(* CODESYS project PRG1545637205.project

Project tree, tasks and I/O mapping:
  Device : CODESYS Control for Raspberry Pi, 3S - Smart Software Solutions GmbH, version 3.5.7.10
    application Application
      libraries: Standard, * (System); SysSocket, 3.5.9.0 (System); SysSem, 3.5.5.0 (System); SysCom, 3.5.5.0 (System); Util, 3.5.11.0 (System); MQTT Client Library, 3.5.0.0 (Stefan Roßmann Engineering Solutions); SysTimeRtc, * (System)
      task MainTask (cyclic, interval t#20ms, priority 1) calls PLC_PRG, Cement_PRG, Automode, Formula, LimeSand, Mixer_PRG, Logger
      task VISU_TASK (cyclic, interval 100 ms, priority 31) calls VisuElems.Visu_Prg
      program PLC_PRG [ST]
      vis/
        visualisation Visualization
        visualisation formula
        visualisation packing
        visualisation lime
        visualisation cement
        visualisation mixer
        visualisation dust
        visualisation other
        visualisation cement_1
        visualisation cement_0
        visualisation cement_2
        visualisation lime_0
        visualisation lime_1
        visualisation lime_3
        visualisation lime_2
        visualisation cement_3
        visualisation mixer_0
        visualisation mixer_1
        visualisation mixer_2
        visualisation mixer_3
        visualisation packing_0
        visualisation packing_3
        visualisation packing_2
        visualisation packing_1
      function block INVT_AO [LD]
      function block Constancheck [ST]
      function block ParamAdjust [ST]
      program LimeSand [LD]
      function block interupt [LD]
      function block Alarm [ST]
      program Automode [LD]
      function block BAYKON [LD]
      program Cement_PRG [LD]
      program Formula [LD]
      function block Formula_Loader [ST]
      function block PulseHold [LD]
      function block screw_speed [ST]
      program Mixer_PRG [LD]
      function block Cycletime [LD]
      MYSQL/
        DUTs/
          data type SHA1Context
          data type MySql_FieldInfo
          data type MySql_FieldTypes
          data type MySql_ResultSet
          data type MySql_ServerInfo
        private/
          SHA/
            function SHA1Hex2String [ST]
            function SHA1Input [ST]
            function SHA1PadMessage [ST]
            function SHA1ProcessMessageBlock [ST]
            function SHA1Reset [ST]
            function SHA1Result [ST]
            function SHA1Version [ST]
            function SHA1 [ST]
          function MySql_Close [ST]
          function block MySql_Context [ST]
          function MySql_Scramble [ST]
        public/
          function MySql_GetStringValue [ST]
          function MySql_Version [ST]
          function block MySql_Execute [ST]
          function block MySql_Login [ST]
          function block MySql_Logout [ST]
          function block MySql_Query [ST]
      global variables GVL_MYSQL
      function block DC [LD]
      program Logger [ST]
    SoftMotion General Axis Pool
    I²C
    SPI
    GPIOs_A_B : GPIOs A/B, 3S - Smart Software Solutions GmbH, version 1.1.1.10
        unmapped channels: digital inputs (GPIO0..GPIO31), digital outputs (GPIO0..GPIO31)
    Onewire
    Camera device
      <Empty>
    Ethernet : Ethernet, 3S - Smart Software Solutions GmbH, version 3.5.10.0
      Modbus_TCP_Master : Modbus TCP Master, 3S - Smart Software Solutions GmbH, version 3.5.10.0
          settings: AutoReconnect = TRUE
        WAGO_170 : Modbus TCP Slave, 3S - Smart Software Solutions GmbH, version 3.5.10.0
            settings: IPAddress = [192, 168, 100, 170]; Channel 0.Function Code = 2; Channel 0.Read Offset = 16#0000; Channel 0.Read Length = 128; Channel 0.Write Offset = 0; Channel 0.Write Length = 0; Channel 0.Cycle Time = 100; Channel 1.Function Code = 3; Channel 1.Read Offset = 16#0000; Channel 1.Read Length = 8; Channel 1.Write Offset = 0; Channel 1.Write Length = 0; Channel 1.Cycle Time = 100; Channel 2.Function Code = 15; Channel 2.Read Offset = 0; Channel 2.Read Length = 0; Channel 2.Write Offset = 16#0000; Channel 2.Write Length = 80; Channel 2.Cycle Time = 100; Channel 3.Function Code = 16; Channel 3.Read Offset = 0; Channel 3.Read Length = 0; Channel 3.Write Offset = 16#0000; Channel 3.Write Length = 4; Channel 3.Cycle Time = 100
            input  DI : ARRAY[0..15] OF BYTE  // Channel 0
            input  DI120 : BYTE  // Channel 0.Channel 0
            input  DI121 : BOOL  // Channel 0.Channel 0.Bit0
            input  DI122 : BOOL  // Channel 0.Channel 0.Bit1
            input  DI123 : BOOL  // Channel 0.Channel 0.Bit2
            input  DI124 : BOOL  // Channel 0.Channel 0.Bit3
            input  DI125 : BOOL  // Channel 0.Channel 0.Bit4
            input  DI126 : BOOL  // Channel 0.Channel 0.Bit5
            input  DI127 : BOOL  // Channel 0.Channel 0.Bit6
            input  DI128 : BOOL  // Channel 0.Channel 0.Bit7
            input  DI130 : BYTE  // Channel 0.Channel 0
            input  DI131 : BOOL  // Channel 0.Channel 0.Bit0
            input  DI132 : BOOL  // Channel 0.Channel 0.Bit1
            input  DI133 : BOOL  // Channel 0.Channel 0.Bit2
            input  DI134 : BOOL  // Channel 0.Channel 0.Bit3
            input  DI135 : BOOL  // Channel 0.Channel 0.Bit4
            input  DI136 : BOOL  // Channel 0.Channel 0.Bit5
            input  DI137 : BOOL  // Channel 0.Channel 0.Bit6
            input  DI138 : BOOL  // Channel 0.Channel 0.Bit7
            input  DI140 : BYTE  // Channel 0.Channel 0
            input  DI141 : BOOL  // Channel 0.Channel 0.Bit0
            input  DI142 : BOOL  // Channel 0.Channel 0.Bit1
            input  DI143 : BOOL  // Channel 0.Channel 0.Bit2
            input  DI144 : BOOL  // Channel 0.Channel 0.Bit3
            input  DI145 : BOOL  // Channel 0.Channel 0.Bit4
            input  DI146 : BOOL  // Channel 0.Channel 0.Bit5
            input  DI147 : BOOL  // Channel 0.Channel 0.Bit6
            input  DI148 : BOOL  // Channel 0.Channel 0.Bit7
            input  DI150 : BYTE  // Channel 0.Channel 0
            input  DI151 : BOOL  // Channel 0.Channel 0.Bit0
            input  DI152 : BOOL  // Channel 0.Channel 0.Bit1
            input  DI153 : BOOL  // Channel 0.Channel 0.Bit2
            input  DI154 : BOOL  // Channel 0.Channel 0.Bit3
            input  DI155 : BOOL  // Channel 0.Channel 0.Bit4
            input  DI156 : BOOL  // Channel 0.Channel 0.Bit5
            input  DI157 : BOOL  // Channel 0.Channel 0.Bit6
            input  DI158 : BOOL  // Channel 0.Channel 0.Bit7
            input  DI160 : BYTE  // Channel 0.Channel 0
            input  DI161 : BOOL  // Channel 0.Channel 0.Bit0
            input  DI162 : BOOL  // Channel 0.Channel 0.Bit1
            input  DI163 : BOOL  // Channel 0.Channel 0.Bit2
            input  DI164 : BOOL  // Channel 0.Channel 0.Bit3
            input  DI165 : BOOL  // Channel 0.Channel 0.Bit4
            input  DI166 : BOOL  // Channel 0.Channel 0.Bit5
            input  DI167 : BOOL  // Channel 0.Channel 0.Bit6
            input  DI168 : BOOL  // Channel 0.Channel 0.Bit7
            input  DI170 : BYTE  // Channel 0.Channel 0
            input  DI171 : BOOL  // Channel 0.Channel 0.Bit0
            input  DI172 : BOOL  // Channel 0.Channel 0.Bit1
            input  DI173 : BOOL  // Channel 0.Channel 0.Bit2
            input  DI174 : BOOL  // Channel 0.Channel 0.Bit3
            input  DI175 : BOOL  // Channel 0.Channel 0.Bit4
            input  DI176 : BOOL  // Channel 0.Channel 0.Bit5
            input  DI177 : BOOL  // Channel 0.Channel 0.Bit6
            input  DI178 : BOOL  // Channel 0.Channel 0.Bit7
            input  DI180 : BYTE  // Channel 0.Channel 0
            input  DI181 : BOOL  // Channel 0.Channel 0.Bit0
            input  DI182 : BOOL  // Channel 0.Channel 0.Bit1
            input  DI183 : BOOL  // Channel 0.Channel 0.Bit2
            input  DI184 : BOOL  // Channel 0.Channel 0.Bit3
            input  DI185 : BOOL  // Channel 0.Channel 0.Bit4
            input  DI186 : BOOL  // Channel 0.Channel 0.Bit5
            input  DI187 : BOOL  // Channel 0.Channel 0.Bit6
            input  DI188 : BOOL  // Channel 0.Channel 0.Bit7
            input  DI190 : BYTE  // Channel 0.Channel 0
            input  DI191 : BOOL  // Channel 0.Channel 0.Bit0
            input  DI192 : BOOL  // Channel 0.Channel 0.Bit1
            input  DI193 : BOOL  // Channel 0.Channel 0.Bit2
            input  DI194 : BOOL  // Channel 0.Channel 0.Bit3
            input  DI195 : BOOL  // Channel 0.Channel 0.Bit4
            input  DI196 : BOOL  // Channel 0.Channel 0.Bit5
            input  DI197 : BOOL  // Channel 0.Channel 0.Bit6
            input  DI198 : BOOL  // Channel 0.Channel 0.Bit7
            input  DI200 : BYTE  // Channel 0.Channel 0
            input  DI201 : BOOL  // Channel 0.Channel 0.Bit0
            input  DI202 : BOOL  // Channel 0.Channel 0.Bit1
            input  DI203 : BOOL  // Channel 0.Channel 0.Bit2
            input  DI204 : BOOL  // Channel 0.Channel 0.Bit3
            input  DI205 : BOOL  // Channel 0.Channel 0.Bit4
            input  DI206 : BOOL  // Channel 0.Channel 0.Bit5
            input  DI207 : BOOL  // Channel 0.Channel 0.Bit6
            input  DI208 : BOOL  // Channel 0.Channel 0.Bit7
            input  DI210 : BYTE  // Channel 0.Channel 0
            input  DI211 : BOOL  // Channel 0.Channel 0.Bit0
            input  DI212 : BOOL  // Channel 0.Channel 0.Bit1
            input  DI213 : BOOL  // Channel 0.Channel 0.Bit2
            input  DI214 : BOOL  // Channel 0.Channel 0.Bit3
            input  DI215 : BOOL  // Channel 0.Channel 0.Bit4
            input  DI216 : BOOL  // Channel 0.Channel 0.Bit5
            input  DI217 : BOOL  // Channel 0.Channel 0.Bit6
            input  DI218 : BOOL  // Channel 0.Channel 0.Bit7
            input  DI220 : BYTE  // Channel 0.Channel 0
            input  DI221 : BOOL  // Channel 0.Channel 0.Bit0
            input  DI222 : BOOL  // Channel 0.Channel 0.Bit1
            input  DI223 : BOOL  // Channel 0.Channel 0.Bit2
            input  DI224 : BOOL  // Channel 0.Channel 0.Bit3
            input  DI225 : BOOL  // Channel 0.Channel 0.Bit4
            input  DI226 : BOOL  // Channel 0.Channel 0.Bit5
            input  DI227 : BOOL  // Channel 0.Channel 0.Bit6
            input  DI228 : BOOL  // Channel 0.Channel 0.Bit7
            input  DI230 : BYTE  // Channel 0.Channel 0
            input  DI231 : BOOL  // Channel 0.Channel 0.Bit0
            input  DI232 : BOOL  // Channel 0.Channel 0.Bit1
            input  DI233 : BOOL  // Channel 0.Channel 0.Bit2
            input  DI234 : BOOL  // Channel 0.Channel 0.Bit3
            input  DI235 : BOOL  // Channel 0.Channel 0.Bit4
            input  DI236 : BOOL  // Channel 0.Channel 0.Bit5
            input  DI237 : BOOL  // Channel 0.Channel 0.Bit6
            input  DI238 : BOOL  // Channel 0.Channel 0.Bit7
            input  DI240 : BYTE  // Channel 0.Channel 0
            input  DI241 : BOOL  // Channel 0.Channel 0.Bit0
            input  DI242 : BOOL  // Channel 0.Channel 0.Bit1
            input  DI243 : BOOL  // Channel 0.Channel 0.Bit2
            input  DI244 : BOOL  // Channel 0.Channel 0.Bit3
            input  DI245 : BOOL  // Channel 0.Channel 0.Bit4
            input  DI246 : BOOL  // Channel 0.Channel 0.Bit5
            input  DI247 : BOOL  // Channel 0.Channel 0.Bit6
            input  DI248 : BOOL  // Channel 0.Channel 0.Bit7
            input  DI250 : BYTE  // Channel 0.Channel 0
            input  DI251 : BOOL  // Channel 0.Channel 0.Bit0
            input  DI252 : BOOL  // Channel 0.Channel 0.Bit1
            input  DI253 : BOOL  // Channel 0.Channel 0.Bit2
            input  DI254 : BOOL  // Channel 0.Channel 0.Bit3
            input  DI255 : BOOL  // Channel 0.Channel 0.Bit4
            input  DI256 : BOOL  // Channel 0.Channel 0.Bit5
            input  DI257 : BOOL  // Channel 0.Channel 0.Bit6
            input  DI258 : BOOL  // Channel 0.Channel 0.Bit7
            input  DI260 : BYTE  // Channel 0.Channel 0
            input  DI261 : BOOL  // Channel 0.Channel 0.Bit0
            input  DI262 : BOOL  // Channel 0.Channel 0.Bit1
            input  DI263 : BOOL  // Channel 0.Channel 0.Bit2
            input  DI264 : BOOL  // Channel 0.Channel 0.Bit3
            input  DI265 : BOOL  // Channel 0.Channel 0.Bit4
            input  DI266 : BOOL  // Channel 0.Channel 0.Bit5
            input  DI267 : BOOL  // Channel 0.Channel 0.Bit6
            input  DI268 : BOOL  // Channel 0.Channel 0.Bit7
            input  DI270 : BYTE  // Channel 0.Channel 0
            input  DI271 : BOOL  // Channel 0.Channel 0.Bit0
            input  DI272 : BOOL  // Channel 0.Channel 0.Bit1
            input  DI273 : BOOL  // Channel 0.Channel 0.Bit2
            input  DI274 : BOOL  // Channel 0.Channel 0.Bit3
            input  DI275 : BOOL  // Channel 0.Channel 0.Bit4
            input  DI276 : BOOL  // Channel 0.Channel 0.Bit5
            input  DI277 : BOOL  // Channel 0.Channel 0.Bit6
            input  DI278 : BOOL  // Channel 0.Channel 0.Bit7
            input  AI : ARRAY[0..7] OF WORD  // Channel 1
            input  AI281 : WORD  // Channel 1.Channel 1
            input  AI282 : WORD  // Channel 1.Channel 1
            input  AI283 : WORD  // Channel 1.Channel 1
            input  AI284 : WORD  // Channel 1.Channel 1
            input  AI291 : WORD  // Channel 1.Channel 1
            input  AI292 : WORD  // Channel 1.Channel 1
            input  AI293 : WORD  // Channel 1.Channel 1
            input  AI294 : WORD  // Channel 1.Channel 1
            output DO311 : BOOL  // Channel 2.Channel 2.Bit0
            output DO312 : BOOL  // Channel 2.Channel 2.Bit1
            output DO313 : BOOL  // Channel 2.Channel 2.Bit2
            output DO314 : BOOL  // Channel 2.Channel 2.Bit3
            output DO315 : BOOL  // Channel 2.Channel 2.Bit4
            output DO316 : BOOL  // Channel 2.Channel 2.Bit5
            output DO317 : BOOL  // Channel 2.Channel 2.Bit6
            output DO318 : BOOL  // Channel 2.Channel 2.Bit7
            output DO321 : BOOL  // Channel 2.Channel 2.Bit0
            output DO322 : BOOL  // Channel 2.Channel 2.Bit1
            output DO323 : BOOL  // Channel 2.Channel 2.Bit2
            output DO324 : BOOL  // Channel 2.Channel 2.Bit3
            output DO325 : BOOL  // Channel 2.Channel 2.Bit4
            output DO326 : BOOL  // Channel 2.Channel 2.Bit5
            output DO327 : BOOL  // Channel 2.Channel 2.Bit6
            output DO328 : BOOL  // Channel 2.Channel 2.Bit7
            output DO331 : BOOL  // Channel 2.Channel 2.Bit0
            output DO332 : BOOL  // Channel 2.Channel 2.Bit1
            output DO333 : BOOL  // Channel 2.Channel 2.Bit2
            output DO334 : BOOL  // Channel 2.Channel 2.Bit3
            output DO335 : BOOL  // Channel 2.Channel 2.Bit4
            output DO336 : BOOL  // Channel 2.Channel 2.Bit5
            output DO337 : BOOL  // Channel 2.Channel 2.Bit6
            output DO338 : BOOL  // Channel 2.Channel 2.Bit7
            output DO341 : BOOL  // Channel 2.Channel 2.Bit0
            output DO342 : BOOL  // Channel 2.Channel 2.Bit1
            output DO343 : BOOL  // Channel 2.Channel 2.Bit2
            output DO344 : BOOL  // Channel 2.Channel 2.Bit3
            output DO345 : BOOL  // Channel 2.Channel 2.Bit4
            output DO346 : BOOL  // Channel 2.Channel 2.Bit5
            output DO347 : BOOL  // Channel 2.Channel 2.Bit6
            output DO348 : BOOL  // Channel 2.Channel 2.Bit7
            output DO351 : BOOL  // Channel 2.Channel 2.Bit0
            output DO352 : BOOL  // Channel 2.Channel 2.Bit1
            output DO353 : BOOL  // Channel 2.Channel 2.Bit2
            output DO354 : BOOL  // Channel 2.Channel 2.Bit3
            output DO355 : BOOL  // Channel 2.Channel 2.Bit4
            output DO356 : BOOL  // Channel 2.Channel 2.Bit5
            output DO357 : BOOL  // Channel 2.Channel 2.Bit6
            output DO358 : BOOL  // Channel 2.Channel 2.Bit7
            output DO371 : BOOL  // Channel 2.Channel 2.Bit0
            output DO372 : BOOL  // Channel 2.Channel 2.Bit1
            output DO373 : BOOL  // Channel 2.Channel 2.Bit2
            output DO374 : BOOL  // Channel 2.Channel 2.Bit3
            output DO375 : BOOL  // Channel 2.Channel 2.Bit4
            output DO376 : BOOL  // Channel 2.Channel 2.Bit5
            output DO377 : BOOL  // Channel 2.Channel 2.Bit6
            output DO378 : BOOL  // Channel 2.Channel 2.Bit7
            output DO381 : BOOL  // Channel 2.Channel 2.Bit0
            output DO382 : BOOL  // Channel 2.Channel 2.Bit1
            output DO383 : BOOL  // Channel 2.Channel 2.Bit2
            output DO384 : BOOL  // Channel 2.Channel 2.Bit3
            output DO385 : BOOL  // Channel 2.Channel 2.Bit4
            output DO386 : BOOL  // Channel 2.Channel 2.Bit5
            output DO387 : BOOL  // Channel 2.Channel 2.Bit6
            output DO388 : BOOL  // Channel 2.Channel 2.Bit7
            output DO391 : BOOL  // Channel 2.Channel 2.Bit0
            output DO392 : BOOL  // Channel 2.Channel 2.Bit1
            output DO393 : BOOL  // Channel 2.Channel 2.Bit2
            output DO394 : BOOL  // Channel 2.Channel 2.Bit3
            output DO395 : BOOL  // Channel 2.Channel 2.Bit4
            output DO396 : BOOL  // Channel 2.Channel 2.Bit5
            output DO397 : BOOL  // Channel 2.Channel 2.Bit6
            output DO398 : BOOL  // Channel 2.Channel 2.Bit7
            output DO401 : BOOL  // Channel 2.Channel 2.Bit0
            output DO402 : BOOL  // Channel 2.Channel 2.Bit1
            output DO403 : BOOL  // Channel 2.Channel 2.Bit2
            output DO404 : BOOL  // Channel 2.Channel 2.Bit3
            output DO405 : BOOL  // Channel 2.Channel 2.Bit4
            output DO406 : BOOL  // Channel 2.Channel 2.Bit5
            output DO407 : BOOL  // Channel 2.Channel 2.Bit6
            output DO408 : BOOL  // Channel 2.Channel 2.Bit7
            output DO411 : BOOL  // Channel 2.Channel 2.Bit0
            output DO412 : BOOL  // Channel 2.Channel 2.Bit1
            output DO413 : BOOL  // Channel 2.Channel 2.Bit2
            output DO414 : BOOL  // Channel 2.Channel 2.Bit3
            output DO415 : BOOL  // Channel 2.Channel 2.Bit4
            output DO416 : BOOL  // Channel 2.Channel 2.Bit5
            output DO417 : BOOL  // Channel 2.Channel 2.Bit6
            output DO418 : BOOL  // Channel 2.Channel 2.Bit7
            output AO431 : WORD  // Channel 3.Channel 3
            output AO432 : WORD  // Channel 3.Channel 3
            output AO441 : WORD  // Channel 3.Channel 3
            output AO442 : WORD  // Channel 3.Channel 3
            unmapped channels: Channel 2, Channel 3
        Baykon_171 : Modbus TCP Slave, 3S - Smart Software Solutions GmbH, version 3.5.10.0
            settings: Unit-ID = 1; IPAddress = [192, 168, 100, 171]; Channel 0.Function Code = 3; Channel 0.Read Offset = 16#0000; Channel 0.Read Length = 7; Channel 0.Write Offset = 0; Channel 0.Write Length = 0; Channel 0.Cycle Time = 100
            input  cem1 : WORD  // Channel 0.Channel 0
            input  cem2 : WORD  // Channel 0.Channel 0
            input  cem3 : WORD  // Channel 0.Channel 0
            input  cem4 : WORD  // Channel 0.Channel 0
            input  cem5 : WORD  // Channel 0.Channel 0
            input  cem6 : WORD  // Channel 0.Channel 0
            input  cem7 : WORD  // Channel 0.Channel 0
            unmapped channels: Channel 0
        Baykon_172 : Modbus TCP Slave, 3S - Smart Software Solutions GmbH, version 3.5.10.0
            settings: Unit-ID = 1; IPAddress = [192, 168, 100, 172]; Channel 0.Function Code = 3; Channel 0.Read Offset = 16#0000; Channel 0.Read Length = 7; Channel 0.Write Offset = 0; Channel 0.Write Length = 0; Channel 0.Cycle Time = 100
            input  lime1 : WORD  // Channel 0.Channel 0
            input  lime2 : WORD  // Channel 0.Channel 0
            input  lime3 : WORD  // Channel 0.Channel 0
            input  lime4 : WORD  // Channel 0.Channel 0
            input  lime5 : WORD  // Channel 0.Channel 0
            input  lime6 : WORD  // Channel 0.Channel 0
            input  lime7 : WORD  // Channel 0.Channel 0
            unmapped channels: Channel 0
  libraries: VisuSymbols, 3.5.10.0 (System)
  text list GlobalTextList
*)

// Device/Application/MYSQL/DUTs/SHA1Context
TYPE SHA1Context :
(* This structure will hold context information for the hashing operation *)
  STRUCT
	Message_Digest : ARRAY [0..4] OF DWORD ;(* Message Digest (output)          *)
    Length_Low  : DWORD;        			(* Message length in bits           *)
    Length_High : DWORD;       				(* Message length in bits           *)
    Message_Block : ARRAY [0..63] OF BYTE; 	(* 512-bit message blocks      *)
    Message_Block_Index : INT;    			(* Index into message block array   *)
    Computed : BOOL;               			(* Is the digest computed?          *)
    Corrupted: BOOL;              			(* Is the message digest corruped?  *)
  END_STRUCT
END_TYPE

// Device/Application/MYSQL/DUTs/MySql_FieldInfo
TYPE MySql_FieldInfo :
(* This structure contains detail informations about each "column" or "data field" in a result set *)
  STRUCT
	sName : STRING(gcMySql_dwMaxIdentifierLength);
	udiLength : UDINT;
	eType : MySql_FieldTypes;
	wFlags : WORD;
	bDecimals : BYTE;
  END_STRUCT
END_TYPE

(*
VERSION 4.1
 Bytes                      Name
 -----                      ----
 n (Length Coded String)    catalog
 n (Length Coded String)    db
 n (Length Coded String)    table
 n (Length Coded String)    org_table
 n (Length Coded String)    name
 n (Length Coded String)    org_name
 1                          (filler)
 2                          charsetnr
 4                          length
 1                          type
 2                          flags
 1                          decimals
 2                          (filler), always 0x00
 n (Length Coded Binary)    default


length:                  Length of column, according to the definition.
                         Also known as "display length". The value given
                         here may be larger than the actual length, for
                         example an instance of a VARCHAR(2) column may
                         have only 1 character in it.

type:                    The code for the column's data type. Also known as
                         "enum_field_type". The possible values at time of
                         writing (taken from  include/mysql_com.h), in hexadecimal:
                         0x00   FIELD_TYPE_DECIMAL
                         0x01   FIELD_TYPE_TINY
                         0x02   FIELD_TYPE_SHORT
                         0x03   FIELD_TYPE_LONG
                         0x04   FIELD_TYPE_FLOAT
                         0x05   FIELD_TYPE_DOUBLE
                         0x06   FIELD_TYPE_NULL
                         0x07   FIELD_TYPE_TIMESTAMP
                         0x08   FIELD_TYPE_LONGLONG
                         0x09   FIELD_TYPE_INT24
                         0x0a   FIELD_TYPE_DATE
                         0x0b   FIELD_TYPE_TIME
                         0x0c   FIELD_TYPE_DATETIME
                         0x0d   FIELD_TYPE_YEAR
                         0x0e   FIELD_TYPE_NEWDATE
                         0x0f   FIELD_TYPE_VARCHAR (new in MySQL 5.0)
                         0x10   FIELD_TYPE_BIT (new in MySQL 5.0)
                         0xf6   FIELD_TYPE_NEWDECIMAL (new in MYSQL 5.0)
                         0xf7   FIELD_TYPE_ENUM
                         0xf8   FIELD_TYPE_SET
                         0xf9   FIELD_TYPE_TINY_BLOB
                         0xfa   FIELD_TYPE_MEDIUM_BLOB
                         0xfb   FIELD_TYPE_LONG_BLOB
                         0xfc   FIELD_TYPE_BLOB
                         0xfd   FIELD_TYPE_VAR_STRING
                         0xfe   FIELD_TYPE_STRING
                         0xff   FIELD_TYPE_GEOMETRY

flags:                   The possible flag values at time of
                         writing (taken from  include/mysql_com.h), in hexadecimal:
                         0001 NOT_NULL_FLAG
                         0002 PRI_KEY_FLAG
                         0004 UNIQUE_KEY_FLAG
                         0008 MULTIPLE_KEY_FLAG
                         0010 BLOB_FLAG
                         0020 UNSIGNED_FLAG
                         0040 ZEROFILL_FLAG
                         0080 BINARY_FLAG
                         0100 ENUM_FLAG
                         0200 AUTO_INCREMENT_FLAG
                         0400 TIMESTAMP_FLAG
                         0800 SET_FLAG

decimals:                The number of positions after the decimal
                         point if the type is DECIMAL or NUMERIC.
                         Also known as "scale".


*)

// Device/Application/MYSQL/DUTs/MySql_FieldTypes
TYPE MySql_FieldTypes :
(
	MYSQL_TYPE_DECIMAL,
	MYSQL_TYPE_TINY,
	MYSQL_TYPE_SHORT,
	MYSQL_TYPE_LONG,
	MYSQL_TYPE_FLOAT,
	MYSQL_TYPE_DOUBLE,
	MYSQL_TYPE_NULL,
	MYSQL_TYPE_TIMESTAMP,
	MYSQL_TYPE_LONGLONG,
	MYSQL_TYPE_INT24,
	MYSQL_TYPE_DATE,
	MYSQL_TYPE_TIME,
	MYSQL_TYPE_DATETIME,
	MYSQL_TYPE_YEAR,
	MYSQL_TYPE_NEWDATE,
	MYSQL_TYPE_VARCHAR,
	MYSQL_TYPE_BIT,
	MYSQL_TYPE_NEWDECIMAL:=246,
	MYSQL_TYPE_ENUM:=247,
	MYSQL_TYPE_SET:=248,
	MYSQL_TYPE_TINY_BLOB:=249,
	MYSQL_TYPE_MEDIUM_BLOB:=250,
	MYSQL_TYPE_LONG_BLOB:=251,
	MYSQL_TYPE_BLOB:=252,
	MYSQL_TYPE_VAR_STRING:=253,
	MYSQL_TYPE_STRING:=254,
	MYSQL_TYPE_GEOMETRY:=255
);
END_TYPE

// Device/Application/MYSQL/DUTs/MySql_ResultSet
TYPE MySql_ResultSet :
(* This structure contains the response data of a succesful executed SELECT statement in a raw format.
Use function "MySql_GetStringValue()" to access and convert raw data into IEC-STRING.
Afterwarts use IEC-Convert functions "STRING_TO_x" to map data to local PLC-Variables.*) 
  STRUCT
	uiColumnCount : UINT; (* Number of columns in a dataset *)
	astColumns : ARRAY [0..gcMySql_dwMaxColumnCount] OF MySql_FieldInfo; (* Column-Details *)
	uiRowCount : UINT; (* Number of datasets in servers response *)
	abRows : ARRAY [0..gcMySql_dwMaxRowCount] OF ARRAY [0..gcMySql_dwMaxRowSize] OF BYTE; (* Raw datasets *)
  END_STRUCT
END_TYPE

// Device/Application/MYSQL/DUTs/MySql_ServerInfo
TYPE MySql_ServerInfo :
(* This structure keep information about the server.
Information are received with "Handshake-Initialisation-Packet" on LOGIN *)
  STRUCT
	bProtocolVersion : BYTE;
	sServerVersion : STRING;
	dwThreadId	: DWORD;
	abScrambleBuffer : ARRAY [0..20] OF BYTE;
	wServerCapabilities : WORD;
	bServerLanguageId : BYTE;
	wServerStatus : WORD;
  END_STRUCT
END_TYPE
(*
 protocol_version:    The server takes this from PROTOCOL_VERSION
                      in /include/mysql_version.h. Example value = 10.
 
 server_version:      The server takes this from MYSQL_SERVER_VERSION
                      in /include/mysql_version.h. Example value = "4.1.1-alpha".
 
 thread_number:       ID of the server thread for this connection.
 
 scramble_buff:       The password mechanism uses this. The second part are the
                      last 13 bytes.
                      (See "Password functions" section elsewhere in this document.)
 
 server_capabilities: CLIENT_XXX options. The possible flag values at time of
 writing (taken from  include/mysql_com.h):
		  CLIENT_LONG_PASSWORD		     1	/* new more secure passwords */
		  CLIENT_FOUND_ROWS			     2	/* Found instead of affected rows */
		  CLIENT_LONG_FLAG			     4	/* Get all column flags */
		  CLIENT_CONNECT_WITH_DB	     8	/* One can specify db on connect */
		  CLIENT_NO_SCHEMA			    16	/* Don't allow database.table.column */
		  CLIENT_COMPRESS			    32	/* Can use compression protocol */
		  CLIENT_ODBC				    64	/* Odbc client */
		  CLIENT_LOCAL_FILES		   128	/* Can use LOAD DATA LOCAL */
		  CLIENT_IGNORE_SPACE		   256	/* Ignore spaces before '(' */
		  CLIENT_PROTOCOL_41		   512	/* New 4.1 protocol */
		  CLIENT_INTERACTIVE	   	  1024	/* This is an interactive client */
		  CLIENT_SSL              	  2048	/* Switch to SSL after handshake */
		  CLIENT_IGNORE_SIGPIPE   	  4096  /* IGNORE sigpipes */
		  CLIENT_TRANSACTIONS		  8192	/* Client knows about transactions */
		  CLIENT_RESERVED         	 16384  /* Old flag for 4.1 protocol  */
		  CLIENT_SECURE_CONNECTION 	 32768  /* New 4.1 authentication */
		  CLIENT_MULTI_STATEMENTS 	 65536  /* Enable/disable multi-stmt support */
		  CLIENT_MULTI_RESULTS    	131072  /* Enable/disable multi-results */
 
 server_language:     current server character set number
 
 server_status:       SERVER_STATUS_xxx flags: e.g. SERVER_STATUS_AUTOCOMMIT
*)

// Device/Application/GVL_MYSQL
VAR_GLOBAL CONSTANT
	(* Global constants could be modified by hiding with a global constant of the same name in your project *)

	gcMySql_dwMaxColumnCount: DWORD := 15; (* Defines the maximum number of columns in a result set
				this library can process.
	*)

	gcMySql_dwMaxRowCount : DWORD := 40; (* Defines the maximum number of rows in a result set
				this library can process.
	*)

	gcMySql_dwMaxRowSize : DWORD := 500; (* Defines the maximum length (size in bytes) of one row in a result set
				this library can process.
	*)

	gcMySql_xClearResultSetBeforeUse : BOOL := FALSE; (* Clear the "stResultSet" before use(need approximatly 400ms),
				used by function block "MySql_Query".  
	*)

	gcMySql_tResponseCompliedlyReceived : TIME := t#50ms; 	(* Wait time - before processing received response data.
				Used to be shure complied response are received. The Wait time is started with first response package
				and restarted on every received response package. Helpful when dialing with slow servers.
				Used by function block "MySql_Query".  
	*)

	gcMySql_dwMaxIdentifierLength : DWORD := 80; (* Defines the maximum length (size in bytes) of a column name,
				used by structure "MySql_FieldInfo", this library can process.
	*)

	gcMySql_iSqlUpperBound: INT := 10; (* Defines the upper bound of "asSqlStatement",
				used by function blocks "MySql_ExecSql" and "MySql_Query" 
				to provide an SQL statement as "ARRAY [0..UpperBound] OF STRING(Size)".
	*)

	gcMySql_iSqlLength: INT := 100; (* Defines the size in byte of an array element
				of "asSqlStatement", used by function blocks "MySql_ExecSql" and "MySql_Query" 
				to provide an SQL statement as "ARRAY [0..UpperBound] OF STRING(Size)".
	*)

	gcMySql_tTimeOut : TIME := t#10s; 	(* WatchDog time -
				Defines the maximum time a function block is operating in the same stage without progress. 
	*)

	gcMySql_dwTxBufferSize: DWORD := 8000; (* Defines the transmit buffer size
	*)

	gcMySql_dwRxBufferSize: DWORD := 40000; (* Defines the receive buffer size
	*)

	gcMySql_dwMaxPacketSize: DWORD := 1024; (* The maximum number of bytes in a packet for the client.
	*)

	gcMySql_bCharsetNumber : BYTE := 16#08; (*
				+------+--------------------+-------------------+
				| ID   | CHARACTER_SET_NAME | COLLATION_NAME    |
				+------+--------------------+-------------------+
				| 16#08| latin1             | latin1_swedish_ci |
				+------+--------------------+-------------------+
				To operate in the same domain as the server, check 
				"pstMySql^.stServerInfo.bServerLanguage", that the
				server passes in the Handshake Initialization packet
	*)

	gcMySql_wClientFlags : WORD := 16#8601; (* CLIENT_xxx options.

				The list of flags taken from ethereal sniff with server version "5.0.67-community-nt" ):
												
					  CLIENT_LONG_PASSWORD		.... .... .... ...1	| ON  | new more secure passwords */
					  CLIENT_FOUND_ROWS			.... .... .... ..0.	| OFF | Found instead of affected rows */
					  CLIENT_LONG_FLAG			.... .... .... .0..	| OFF | Get all column flags */
					  CLIENT_CONNECT_WITH_DB	.... .... .... 0...	| OFF | One can specify db on connect */
					  CLIENT_NO_SCHEMA			.... .... ...0 ....	| OFF | Don't allow database.table.column */
					  CLIENT_COMPRESS			.... .... ..0. ....	| OFF | Can use compression protocol */
					  CLIENT_ODBC				.... .... .0.. ....	| OFF | Odbc client */
					  CLIENT_LOCAL_FILES		.... .... 0... .... | OFF | Can use LOAD DATA LOCAL */
					  CLIENT_IGNORE_SPACE		.... ...0 .... .... | OFF | Ignore spaces before '(' */
					  CLIENT_PROTOCOL_41		.... ..1. .... .... | ON  | New 4.1 protocol */
					  CLIENT_INTERACTIVE	   	.... .1.. .... .... | ON  | This is an interactive client */
					  CLIENT_SSL              	.... 0... .... .... | OFF | Switch to SSL after handshake */
					  CLIENT_IGNORE_SIGPIPE   	...0 .... .... .... | OFF | IGNORE sigpipes */
					  CLIENT_TRANSACTIONS		..0. .... .... .... | OFF | Client knows about transactions */
					  CLIENT_RESERVED         	.0.. .... .... .... | OFF | Old flag for 4.1 protocol  */
					  CLIENT_SECURE_CONNECTION 	1... .... .... .... | ON  | New 4.1 authentication */

												1... .11. .... ...1 ==> 16#8601

                  Values is in the description of the Handshake
                  Initialisation Packet, for server_capabilities.
                  For some of the bits, the server passed "what
                  it's capable of". The client leaves some of the
                  bits on, adds others, and passes back to the server.
                  One important flag is: whether compression is desired.
                  Another interesting one is CLIENT_CONNECT_WITH_DB,
                  which shows the presence of the optional databasename.
	*)

	gcMySql_wExtClientFlags : WORD := 16#0003; (* Extend CLIENT_xxx options.

					  CLIENT_MULTI_STATEMENTS 	 .... .... .... ...1 | ON  | Enable/disable multi-stmt support */
					  CLIENT_MULTI_RESULTS    	 .... .... .... ..1. | ON  | Enable/disable multi-results */
	*)
END_VAR
VAR_GLOBAL
	gatel: INT := 12;
END_VAR

// Device/Application/PLC_PRG
PROGRAM PLC_PRG
VAR
	lighting1A: BOOL;
	lighting1B: BOOL;
	lighting2A: BOOL;
	lighting2B: BOOL;
	lighting3: BOOL;
	lighting4: BOOL;
	jamON: ParamAdjust;
	jamOFF: ParamAdjust;
	light_on: REAL;
	add_light_on: BOOL;
	sub_light_on: BOOL;
	l1a: BOOL := true;
	l1b: BOOL := true;
	l2a: BOOL := true;
	l2b: BOOL := true;
	l3: BOOL := true;
	l4: BOOL := true;
END_VAR




IF lighting1A = TRUE OR Formula.lampu = TRUE THEN
	l1a := TRUE;
	ELSE
		l1a := FALSE;
END_IF
DO337 := NOT l1a;
IF lighting1B = TRUE OR Formula.lampu = TRUE THEN
	l1b := TRUE;
	ELSE
		l1b := FALSE;
END_IF
DO338 := NOT l1b;
IF lighting2A = TRUE OR Formula.lampu = TRUE THEN
	l2a := TRUE;
	ELSE
		l2a := FALSE;
END_IF
DO341 := NOT l2a;
IF lighting2B = TRUE OR Formula.lampu = TRUE THEN
	l2b := TRUE;
	ELSE
		l2b := FALSE;
END_IF
DO342 := NOT l2b;
IF lighting3 = TRUE OR Formula.lampu = TRUE THEN
	l3 := TRUE;
	ELSE
		l3 := FALSE;
END_IF
DO343 := NOT l3;
IF lighting4 = TRUE OR Formula.lampu = TRUE THEN
	l4 := TRUE;
	ELSE
		l4 := FALSE;
END_IF
DO344 := NOT l4;

END_PROGRAM

// Device/Application/Formula
PROGRAM Formula
VAR
	Formula_Loader_0: Formula_Loader;
	formula_num: INT := 1;
	ParamAdjust_adj_lime: ParamAdjust;
	adj_lime: REAL;
	adj_cement: REAL;
	adj_sand: REAL;
	adj_c_1: REAL;
	adj_c_2: REAL;
	adj_c_3: REAL;
	lime_target: REAL;
	cement_target: REAL;
	sand_target: REAL;
	c_1_target: REAL;
	c_2_target: REAL;
	c_3_target: REAL;
	formula_name: STRING;
	add_lime: BOOL;
	sub_lime: BOOL;
	ParamAdjust_adj_cement: ParamAdjust;
	add_cement: BOOL;
	sub_cement: BOOL;
	ParamAdjust_adj_sand: ParamAdjust;
	add_sand: BOOL;
	sub_sand: BOOL;
	ParamAdjust_adj_c_1: ParamAdjust;
	add_c_1: BOOL;
	sub_c_1: BOOL;
	ParamAdjust_adj_c_3: ParamAdjust;
	ParamAdjust_adj_c_2: ParamAdjust;
	add_c_2: BOOL;
	sub_c_2: BOOL;
	add_c_3: BOOL;
	sub_c_3: BOOL;
	next_formula: BOOL;
	prev_formula: BOOL;
	agitate_time: REAL;
	main_agitator: BOOL;
	right_agitator: BOOL;
	unixtimex: DWORD;
	getrtc: UDINT;
	jam: UDINT;
	hari: UDINT;
	detik: UDINT;
	jam1: UDINT;
	menit: UDINT;
	jamGMT: UDINT;
	jamWIB: UDINT;
	jamfix: UDINT;
	lampu: BOOL;
	jamnyala: INT := 17;
	jammati: INT := 7;
	tomboltambah: BOOL;
	tombolkurang: BOOL;
	tombolkurangmati: BOOL;
	tomboltambahmati: BOOL;
END_VAR
VAR // added by the converter: edge detectors and wires of the graphical bodies
    _rt1, _rt2, _rt3, _rt4, _rt5, _rt6 : R_TRIG;
END_VAR

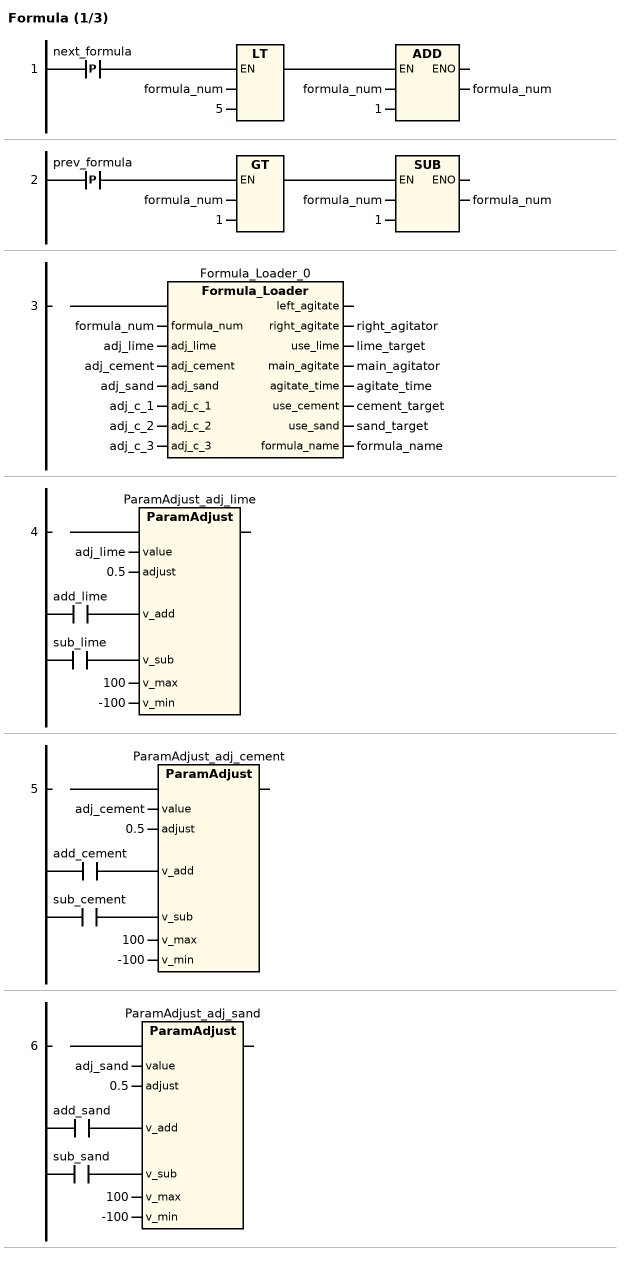
// NETWORK 1
_rt1(CLK := next_formula);
IF _rt1.Q AND formula_num < 5 THEN formula_num := formula_num + 1; END_IF

// NETWORK 2
_rt2(CLK := prev_formula);
IF _rt2.Q AND formula_num > 1 THEN formula_num := formula_num - 1; END_IF

// NETWORK 3
Formula_Loader_0(
    formula_num := formula_num,
    adj_lime := adj_lime,
    adj_cement := adj_cement,
    adj_sand := adj_sand,
    adj_c_1 := adj_c_1,
    adj_c_2 := adj_c_2,
    adj_c_3 := adj_c_3,
    right_agitate => right_agitator,
    use_lime => lime_target,
    main_agitate => main_agitator,
    agitate_time => agitate_time,
    use_cement => cement_target,
    use_sand => sand_target,
    formula_name => formula_name); // Formula_Loader

// NETWORK 4
ParamAdjust_adj_lime(
    value := adj_lime,
    adjust := 0.5,
    v_add := add_lime,
    v_sub := sub_lime,
    v_max := 100,
    v_min := -100); // ParamAdjust

// NETWORK 5
ParamAdjust_adj_cement(
    value := adj_cement,
    adjust := 0.5,
    v_add := add_cement,
    v_sub := sub_cement,
    v_max := 100,
    v_min := -100); // ParamAdjust

// NETWORK 6
ParamAdjust_adj_sand(
    value := adj_sand,
    adjust := 0.5,
    v_add := add_sand,
    v_sub := sub_sand,
    v_max := 100,
    v_min := -100); // ParamAdjust

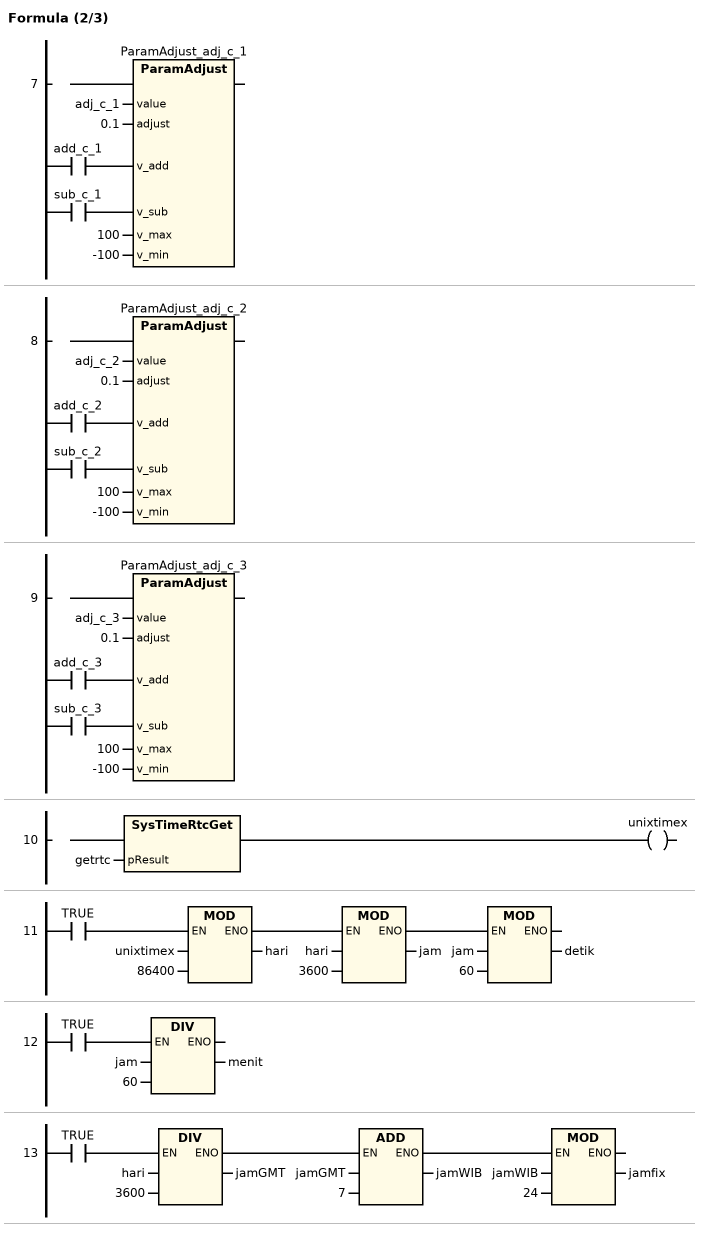
// NETWORK 7
ParamAdjust_adj_c_1(
    value := adj_c_1,
    adjust := 0.1,
    v_add := add_c_1,
    v_sub := sub_c_1,
    v_max := 100,
    v_min := -100); // ParamAdjust

// NETWORK 8
ParamAdjust_adj_c_2(
    value := adj_c_2,
    adjust := 0.1,
    v_add := add_c_2,
    v_sub := sub_c_2,
    v_max := 100,
    v_min := -100); // ParamAdjust

// NETWORK 9
ParamAdjust_adj_c_3(
    value := adj_c_3,
    adjust := 0.1,
    v_add := add_c_3,
    v_sub := sub_c_3,
    v_max := 100,
    v_min := -100); // ParamAdjust

// NETWORK 10
unixtimex := SysTimeRtcGet(pResult := getrtc);

// NETWORK 11
hari := unixtimex MOD 86400;
jam := hari MOD 3600;
detik := jam MOD 60;

// NETWORK 12
menit := jam / 60;

// NETWORK 13
jamGMT := hari / 3600;
jamWIB := jamGMT + 7;
jamfix := jamWIB MOD 24;

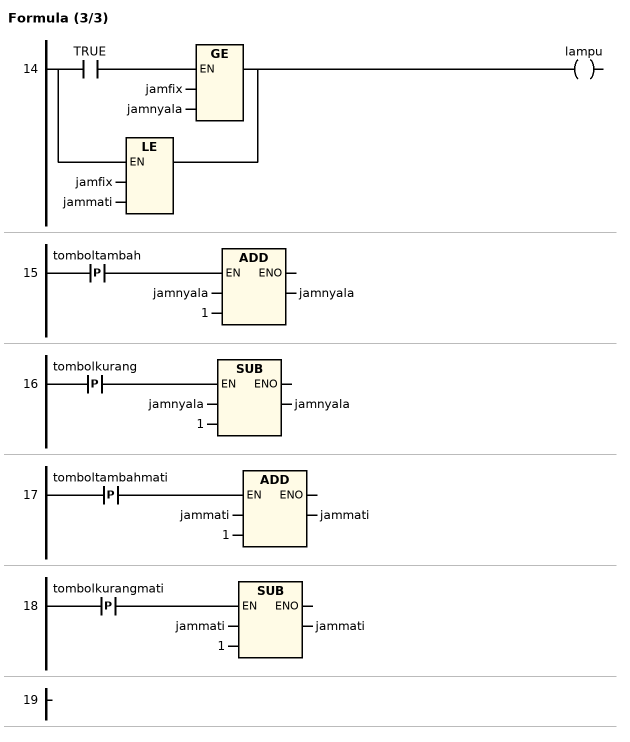
// NETWORK 14
lampu := jamfix >= jamnyala OR jamfix <= jammati;

// NETWORK 15
_rt3(CLK := tomboltambah);
IF _rt3.Q THEN jamnyala := jamnyala + 1; END_IF

// NETWORK 16
_rt4(CLK := tombolkurang);
IF _rt4.Q THEN jamnyala := jamnyala - 1; END_IF

// NETWORK 17
_rt5(CLK := tomboltambahmati);
IF _rt5.Q THEN jammati := jammati + 1; END_IF

// NETWORK 18
_rt6(CLK := tombolkurangmati);
IF _rt6.Q THEN jammati := jammati - 1; END_IF

// NETWORK 19

END_PROGRAM

// Device/Application/Formula_Loader
FUNCTION_BLOCK Formula_Loader
VAR_INPUT
	formula_num: INT := 1;
END_VAR
VAR
	def_lime: REAL;
	def_cement: REAL;
	def_sand: REAL;
	def_c_1: REAL;
	def_c_2: REAL;
	def_c_3: REAL;
END_VAR
VAR_OUTPUT
	left_agitate: BOOL;
	right_agitate: BOOL;
	use_lime: REAL;
	main_agitate: BOOL;
	agitate_time: REAL;
END_VAR
VAR_INPUT
	adj_lime: REAL;
END_VAR
VAR_OUTPUT
	use_cement: REAL;
END_VAR
VAR_INPUT
	adj_cement: REAL;
END_VAR
VAR_OUTPUT
	use_sand: REAL;
END_VAR
VAR_INPUT
	adj_sand: REAL;
END_VAR
VAR
	use_c_1: REAL;
END_VAR
VAR_INPUT
	adj_c_1: REAL;
END_VAR
VAR
	use_c_2: REAL;
END_VAR
VAR_INPUT
	adj_c_2: REAL;
END_VAR
VAR
	use_c_3: REAL;
END_VAR
VAR_INPUT
	adj_c_3: REAL;
END_VAR
VAR_OUTPUT
	formula_name: STRING;
END_VAR

IF formula_num = 1 THEN
	formula_name := 'Thin Bed';
	def_lime := 390;
	def_cement := 185;
	def_sand := 400;
	agitate_time := 150;
	main_agitate := TRUE;
	left_agitate := FALSE;
	right_agitate := FALSE;
	def_c_1 := 1;
	def_c_2 := 0;
	def_c_3 := 0;
END_IF
IF formula_num = 2 THEN
	formula_name := 'Plastering';
	def_lime := 228.52;
	def_cement := 137.11;
	def_sand := 650;
	agitate_time := 150;
	main_agitate := TRUE;
	left_agitate := FALSE;
	right_agitate := FALSE;
	def_c_1 := 100;
	def_c_2 := 100;
	def_c_3 := 100;
END_IF
IF formula_num = 3 THEN
	formula_name := 'Thin Bed (N.C)';
	def_lime := 390;
	def_cement := 0;
	def_sand := 400;
	agitate_time := 150;
	main_agitate := TRUE;
	left_agitate := FALSE;
	right_agitate := FALSE;
	def_c_1 := 100;
	def_c_2 := 100;
	def_c_3 := 100;
END_IF
IF formula_num = 4 THEN
	formula_name := 'Formula No 4';
	def_lime := 400;
	def_cement := 400;
	def_sand := 400;
	agitate_time := 150;
	main_agitate := TRUE;
	left_agitate := FALSE;
	right_agitate := FALSE;
	def_c_1 := 100;
	def_c_2 := 100;
	def_c_3 := 100;
END_IF
IF formula_num = 5 THEN
	formula_name := 'Formula simulasi pake barbel';
	def_lime := 40;
	def_cement := 40;
	def_sand := 40;
	agitate_time := 150;
	main_agitate := TRUE;
	left_agitate := FALSE;
	right_agitate := FALSE;
	def_c_1 := 100;
	def_c_2 := 100;
	def_c_3 := 100;
END_IF
use_lime := def_lime + adj_lime;
use_cement := def_cement + adj_cement;
use_sand := def_sand + adj_sand;
use_c_1 := def_c_1 + adj_c_1;
use_c_2 := def_c_2 + adj_c_2;
use_c_3 := def_c_3 + adj_c_3;

END_FUNCTION_BLOCK

// Device/Application/ParamAdjust
FUNCTION_BLOCK ParamAdjust
VAR
	r_add: r_trig;
	r_sub: r_trig;
END_VAR
VAR_IN_OUT
	value: real := 0;
END_VAR
VAR_INPUT
	adjust: real := 0.1;
	v_add: bool;
	v_sub: BOOL;
	v_max: REAL := 100;
	v_min: REAL := 0;
END_VAR

r_add(CLK:= v_add, Q=> );
r_sub(CLK:= v_sub, Q=> );
IF r_add.Q = TRUE AND value <= v_max THEN
	value := value + adjust; 
END_IF
IF r_sub.Q = TRUE AND value >= v_min THEN
	value := value - adjust; 
END_IF

END_FUNCTION_BLOCK

// Device/Application/Cement_PRG
PROGRAM Cement_PRG
VAR
	start_batch: BOOL;
	BAYKON_cement: BAYKON;
	cement_weight: REAL;
	baykon_system: STRING;
	baykon_data: STRING;
	finish_dosing: BOOL;
	cement_looper: BOOL;
	ParamAdjust_tolerance: ParamAdjust;
	cement_tolerance: REAL := 2;
	add_tolerance: BOOL;
	sub_tolerance: BOOL;
	clean_req: BOOL;
	cement_alarm: STRING;
	auto_cement: BOOL;
	zero_cement: REAL;
	start_weighting: BOOL;
	finish_weighting: BOOL;
	weighting: BOOL;
	//goto DO371
	open_valve: BOOL;
	// go to DO331
	run_screw: BOOL;
	TON_0: TON;
	ParamAdjust_delayrotary: ParamAdjust;
	delay_rotary: REAL := 10;
	add_delayrotary: BOOL;
	sub_delayrotary: BOOL;
	delay_rotaryTime: TIME;
	tmp_rot: TIME;
	// DO313
	run_rotary: BOOL;
	// to DO311and DO312
	run_vibrator: BOOL;
	ParamAdjust_closevalve: ParamAdjust;
	// kg
	closevalve_value: REAL := 0;
	add_close: BOOL;
	sub_close: BOOL;
	interupted: BOOL;
	interupt_fixed: BOOL;
	//go to DI203
	valve_opened: BOOL;
	screw_speed_cement: screw_speed;
	ParamAdjust_slowscrew: ParamAdjust;
	// %
	slow_screw: REAL := 99;
	add_slowscrew: BOOL;
	sub_slowscrew: BOOL;
	ParamAdjust_maxscrew: ParamAdjust;
	// Hz
	max_screw: REAL := 40;
	add_maxscrew: BOOL;
	sub_maxscrew: BOOL;
	ParamAdjust_minscrew: ParamAdjust;
	// Hz
	min_screw: REAL := 20;
	add_minscrew: BOOL;
	sub_minscrew: BOOL;
	ParamAdjust_slowset2: ParamAdjust;
	// %
	slow_screw2: REAL := 99;
	add_slowscrew2: BOOL;
	sub_slowscrew2: BOOL;
	screw_Hz: REAL;
	INVT_AO_screw: INVT_AO;
	screw_fwd: BOOL;
	manual_cement: BOOL;
	auto_screw_Hz: REAL;
	ParamAdjust_screwservice: ParamAdjust;
	// Hz
	service_screw_Hz: REAL := 20;
	add_serviceHz: BOOL;
	sub_serviceHz: BOOL;
	// feedback invt
	screw_run: BOOL;
	service_cement: BOOL := true;
	screw_standby: BOOL;
	screw_rvs: BOOL;
	rvs_relay: BOOL;
	// feedback invt
	screw_fault: BOOL;
	cement_targetfix: REAL;
	ParamAdjust_screwpulse: ParamAdjust;
	// ms
	screwpulse: REAL := 10000;
	add_screwpulse: BOOL;
	sub_screwpulse: BOOL;
	screwpulseTime: TIME;
	PulseHold_Cement: PulseHold;
	// sensor pulse
	screw_rotating: BOOL;
	monit_screw: BOOL;
	TON_monit_screw: TON;
	tmp_monitscrew: TIME;
	ParamAdjust_stoprot: ParamAdjust;
	// kg
	stoprot: REAL := 2;
	add_stoprot: BOOL;
	sub_stoprot: BOOL;
	remaining_cement: REAL;
	stop_rot: BOOL;
	stop_vib: BOOL;
	// cut open valve signal
	close_valve: BOOL;
	end_weighting: BOOL;
	dosing_ready: BOOL;
	dosing_process: BOOL;
	// DO314
	run_rotweight: BOOL;
	manual_weighting: BOOL;
	x_open_valve: BOOL;
	//go to DI204
	valve_closed: BOOL;
	init_cement: BOOL;
	x_run_screw: BOOL;
	// from DI202
	screw_sensor: BOOL;
	screw_contactor: BOOL;
	x_run_rot: BOOL;
	rotary_contactor: BOOL;
	x_run_vib: BOOL;
	vib1_contactor: BOOL;
	vib2_contactor: BOOL;
	TON_protection: TON;
	delay_afterclose: TIME;
	tmp_close: TIME;
	ParamAdjust_afterclose: ParamAdjust;
	afterclose: REAL := 5;
	add_afterclose: BOOL;
	sub_afterclose: BOOL;
	// DO316
	run_vibweight: BOOL;
	manual_dosing: BOOL;
	x_run_rotweight: BOOL;
	x_run_vibweight: BOOL;
	rotweight_contactor: BOOL;
	vibweight_contactor: BOOL;
	manual_finish_dosing: BOOL;
	TON_dosing: TON;
	tank_empty_1: BOOL;
	tmp_dosing: TIME;
	manual_finish_weighting: BOOL;
	delay_rotaryms: REAL;
	afterclosems: REAL;
	x_opened: BOOL;
	x_close_valve: BOOL;
	x_screw: BOOL;
	x_stop_screw: BOOL;
	x_rot: BOOL;
	x_stop_rot: BOOL;
	x_vib: BOOL;
	x_stop_vib: BOOL;
	x_rotweight: BOOL;
	x_stop_rotweight: BOOL;
	auto_cementx: BOOL;
	manual_cementx: BOOL;
	service_cementx: BOOL;
	x_vibweight: BOOL;
	x_stop_vibweight: BOOL;
	check_val: word;
	Constancheck_Cement: Constancheck;
	cement_tank_empty: BOOL;
	Constancheck_beforedosing: Constancheck;
	start_dosing_ok: BOOL;
	Constancheck_beforeweighting: Constancheck;
	start_weighting_ok: BOOL;
	weighting_check: BOOL;
	start_value: REAL;
	dosing_finish: BOOL;
	cement_gross: WORD;
	cekcek: BOOL;
	ceko: BOOL;
	dosing_enable: BOOL;
	weighting_seq: BOOL;
	waiting_mixer: BOOL;
	dosing_seq: BOOL;
	cek_zero_weight: BOOL;
	TON_checkzero: TON;
	zeroTime: TIME := T#1MS;
	tmp_zero: TIME;
	TON_weightingtime: TON;
	weightingTime: TIME := T#60s;
	tmp_weighting: TIME;
	cement_a: REAL;
	cement_amp: REAL;
	start_cement: REAL;
	weighting_time: INT;
	end_cement: REAL;
	weighting_duration: INT;
	start_cement_dosing: REAL;
	end_cement_dosing: REAL;
	dosing_time: INT;
	dosing_duration: INT;
	cement_seq: STRING;
	last_batch: BOOL;
	log_cem: BOOL;
	teslog: BOOL;
	testbaykon: BOOL;
	errc: MB_ErrorCodes;
	baykon_mati: BOOL;
	TON_mati: TON;
	tmpmati: TIME;
	baykon_disconnect: BOOL;
	baykon_dis: BOOL;
	TON_murub: TON;
	tmpmurub: TIME;
END_VAR
VAR // added by the converter: edge detectors and wires of the graphical bodies
    _rt1, _rt2, _rt3, _rt4, _rt5, _rt6, _rt7, _rt8, _rt9, _rt10, _rt11, _rt12, _rt13, _rt14, _rt15, _rt16, _rt17, _rt18, _rt19, _rt20, _rt21, _rt22, _rt23, _rt24, _rt25, _rt26 : R_TRIG;
    _w1, _w2, _w3, _w4, _w5, _w6, _w7, _w8, _w9, _w10, _w11, _w12, _w13, _w14 : BOOL;
    _ft1, _ft2 : F_TRIG;
END_VAR

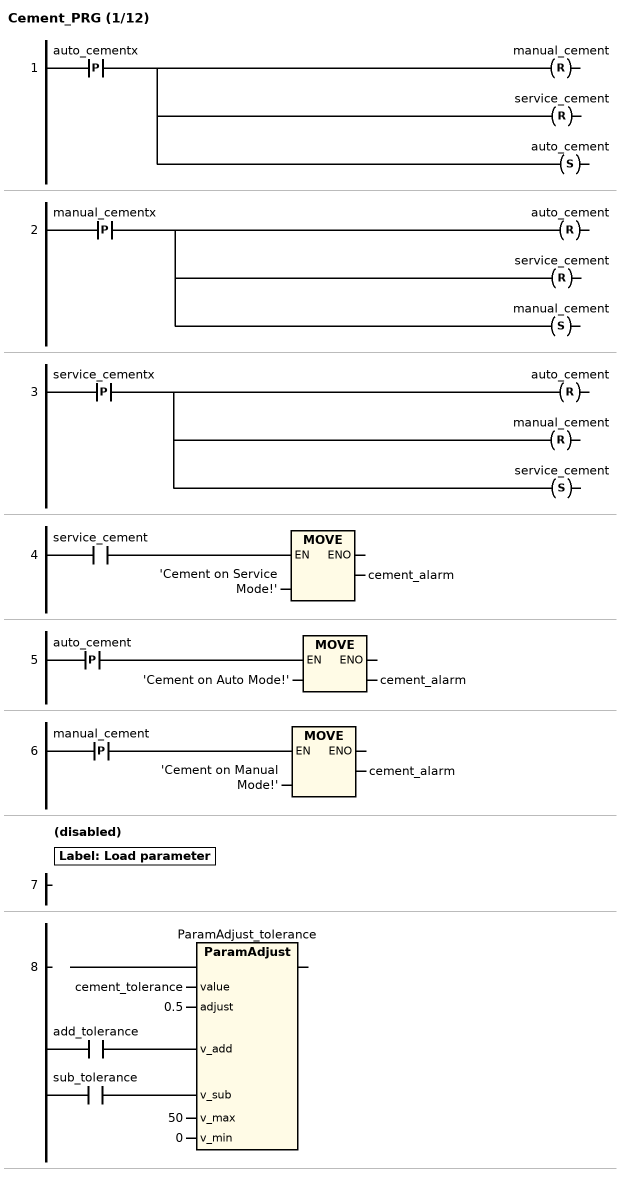
// NETWORK 1
_rt1(CLK := auto_cementx);
manual_cement R= _rt1.Q;
service_cement R= _rt1.Q;
auto_cement S= _rt1.Q;

// NETWORK 2
_rt2(CLK := manual_cementx);
auto_cement R= _rt2.Q;
service_cement R= _rt2.Q;
manual_cement S= _rt2.Q;

// NETWORK 3
_rt3(CLK := service_cementx);
auto_cement R= _rt3.Q;
manual_cement R= _rt3.Q;
service_cement S= _rt3.Q;

// NETWORK 4
IF service_cement THEN cement_alarm := 'Cement on Service Mode!'; END_IF

// NETWORK 5
_rt4(CLK := auto_cement);
IF _rt4.Q THEN cement_alarm := 'Cement on Auto Mode!'; END_IF

// NETWORK 6
_rt5(CLK := manual_cement);
IF _rt5.Q THEN cement_alarm := 'Cement on Manual Mode!'; END_IF

// NETWORK 7 (disabled)
// label: Label: Load parameter

// NETWORK 8
ParamAdjust_tolerance(
    value := cement_tolerance,
    adjust := 0.5,
    v_add := add_tolerance,
    v_sub := sub_tolerance,
    v_max := 50,
    v_min := 0); // ParamAdjust

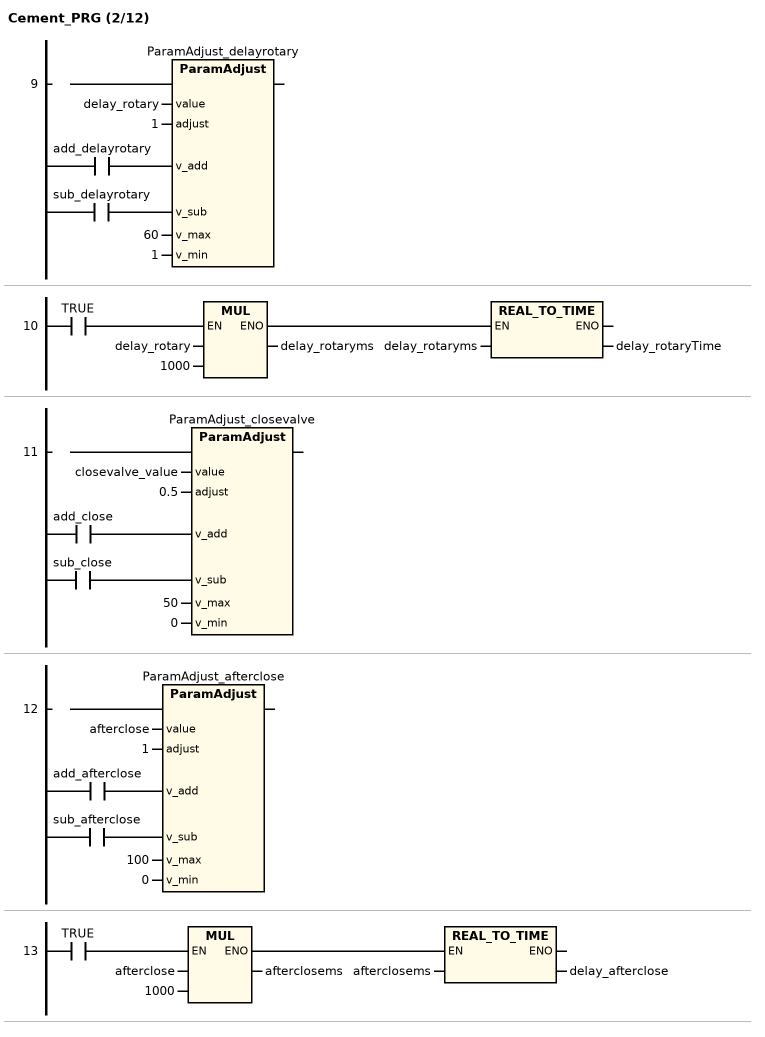
// NETWORK 9
ParamAdjust_delayrotary(
    value := delay_rotary,
    adjust := 1,
    v_add := add_delayrotary,
    v_sub := sub_delayrotary,
    v_max := 60,
    v_min := 1); // ParamAdjust

// NETWORK 10
delay_rotaryms := delay_rotary * 1000;
delay_rotaryTime := REAL_TO_TIME(delay_rotaryms);

// NETWORK 11
ParamAdjust_closevalve(
    value := closevalve_value,
    adjust := 0.5,
    v_add := add_close,
    v_sub := sub_close,
    v_max := 50,
    v_min := 0); // ParamAdjust

// NETWORK 12
ParamAdjust_afterclose(
    value := afterclose,
    adjust := 1,
    v_add := add_afterclose,
    v_sub := sub_afterclose,
    v_max := 100,
    v_min := 0); // ParamAdjust

// NETWORK 13
afterclosems := afterclose * 1000;
delay_afterclose := REAL_TO_TIME(afterclosems);

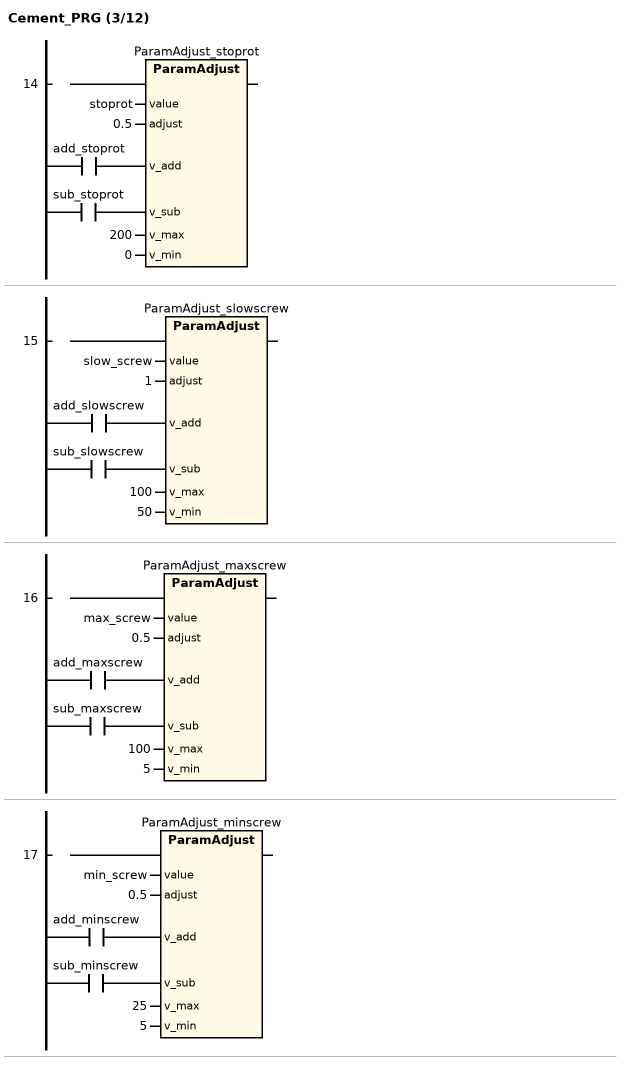
// NETWORK 14
ParamAdjust_stoprot(
    value := stoprot,
    adjust := 0.5,
    v_add := add_stoprot,
    v_sub := sub_stoprot,
    v_max := 200,
    v_min := 0); // ParamAdjust

// NETWORK 15
ParamAdjust_slowscrew(
    value := slow_screw,
    adjust := 1,
    v_add := add_slowscrew,
    v_sub := sub_slowscrew,
    v_max := 100,
    v_min := 50); // ParamAdjust

// NETWORK 16
ParamAdjust_maxscrew(
    value := max_screw,
    adjust := 0.5,
    v_add := add_maxscrew,
    v_sub := sub_maxscrew,
    v_max := 100,
    v_min := 5); // ParamAdjust

// NETWORK 17
ParamAdjust_minscrew(
    value := min_screw,
    adjust := 0.5,
    v_add := add_minscrew,
    v_sub := sub_minscrew,
    v_max := 25,
    v_min := 5); // ParamAdjust

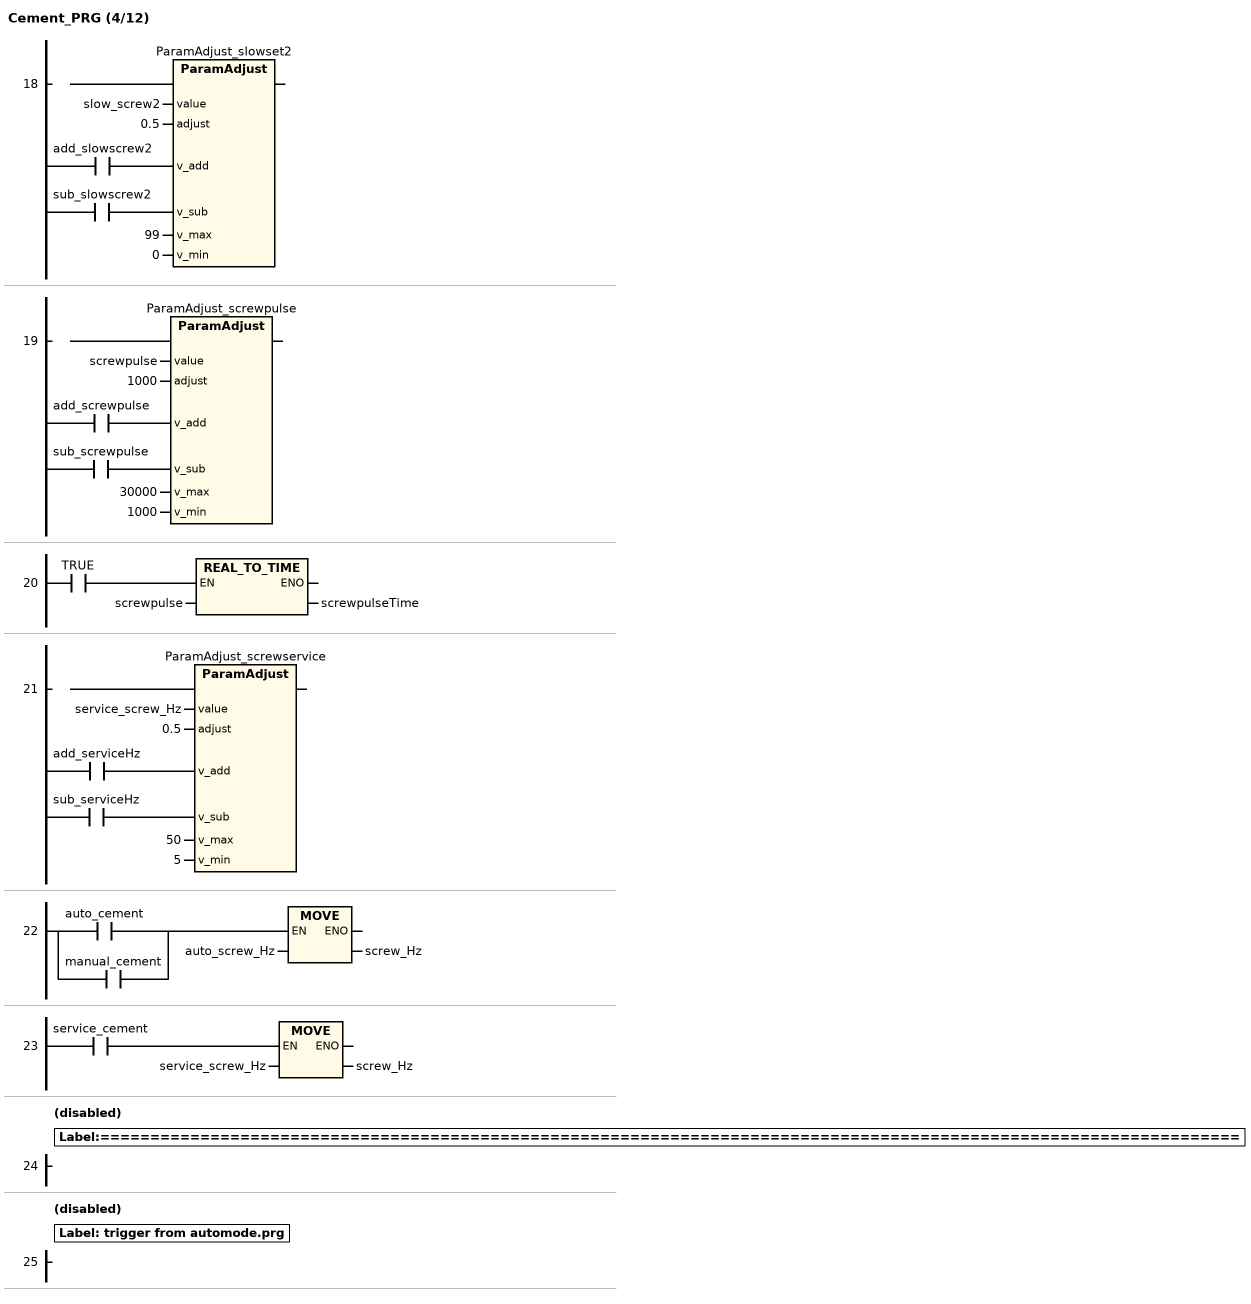
// NETWORK 18
ParamAdjust_slowset2(
    value := slow_screw2,
    adjust := 0.5,
    v_add := add_slowscrew2,
    v_sub := sub_slowscrew2,
    v_max := 99,
    v_min := 0); // ParamAdjust

// NETWORK 19
ParamAdjust_screwpulse(
    value := screwpulse,
    adjust := 1000,
    v_add := add_screwpulse,
    v_sub := sub_screwpulse,
    v_max := 30000,
    v_min := 1000); // ParamAdjust

// NETWORK 20
screwpulseTime := REAL_TO_TIME(screwpulse);

// NETWORK 21
ParamAdjust_screwservice(
    value := service_screw_Hz,
    adjust := 0.5,
    v_add := add_serviceHz,
    v_sub := sub_serviceHz,
    v_max := 50,
    v_min := 5); // ParamAdjust

// NETWORK 22
IF auto_cement OR manual_cement THEN screw_Hz := auto_screw_Hz; END_IF

// NETWORK 23
IF service_cement THEN screw_Hz := service_screw_Hz; END_IF

// NETWORK 24 (disabled)
// label: Label:==================================================================================================================

// NETWORK 25 (disabled)
// label: Label: trigger from automode.prg

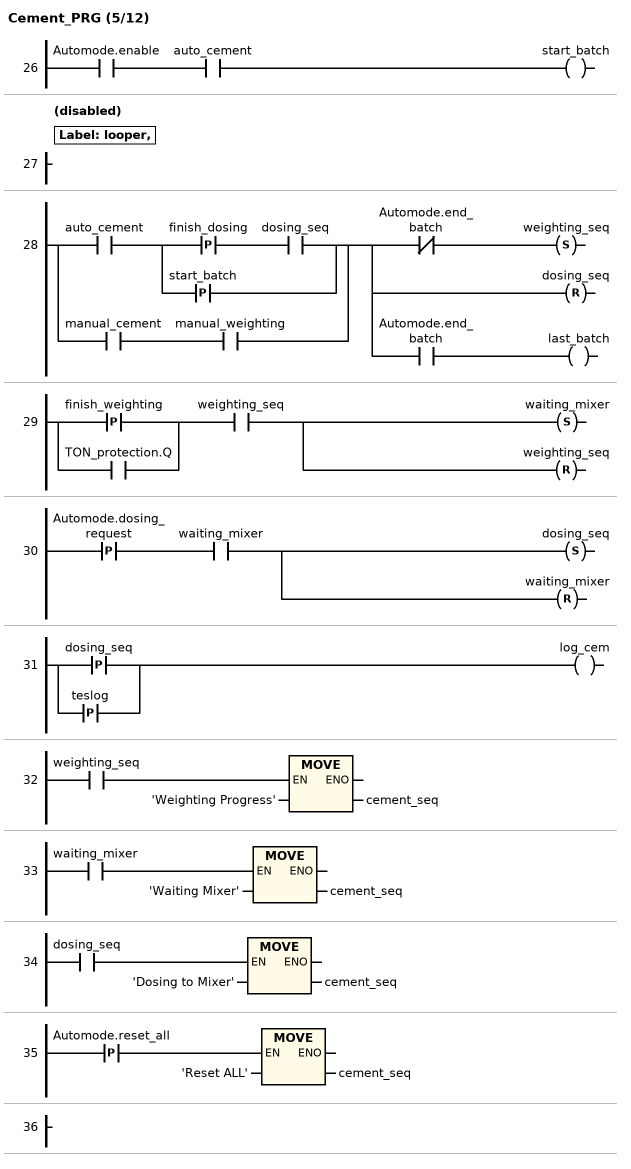
// NETWORK 26
start_batch := Automode.enable AND auto_cement;

// NETWORK 27 (disabled)
// label: Label: looper,

// NETWORK 28
_rt6(CLK := finish_dosing);
_rt7(CLK := start_batch);
_w1 := auto_cement AND (_rt6.Q AND dosing_seq OR _rt7.Q) OR manual_cement AND manual_weighting;
weighting_seq S= _w1 AND NOT Automode.end_batch;
dosing_seq R= _w1;
last_batch := _w1 AND Automode.end_batch;

// NETWORK 29
_rt8(CLK := finish_weighting);
_w2 := (_rt8.Q OR TON_protection.Q) AND weighting_seq;
waiting_mixer S= _w2;
weighting_seq R= _w2;

// NETWORK 30
_rt9(CLK := Automode.dosing_request);
_w3 := _rt9.Q AND waiting_mixer;
dosing_seq S= _w3;
waiting_mixer R= _w3;

// NETWORK 31
_rt10(CLK := dosing_seq);
_rt11(CLK := teslog);
log_cem := _rt10.Q OR _rt11.Q;

// NETWORK 32
IF weighting_seq THEN cement_seq := 'Weighting Progress'; END_IF

// NETWORK 33
IF waiting_mixer THEN cement_seq := 'Waiting Mixer'; END_IF

// NETWORK 34
IF dosing_seq THEN cement_seq := 'Dosing to Mixer'; END_IF

// NETWORK 35
_rt12(CLK := Automode.reset_all);
IF _rt12.Q THEN cement_seq := 'Reset ALL'; END_IF

// NETWORK 36

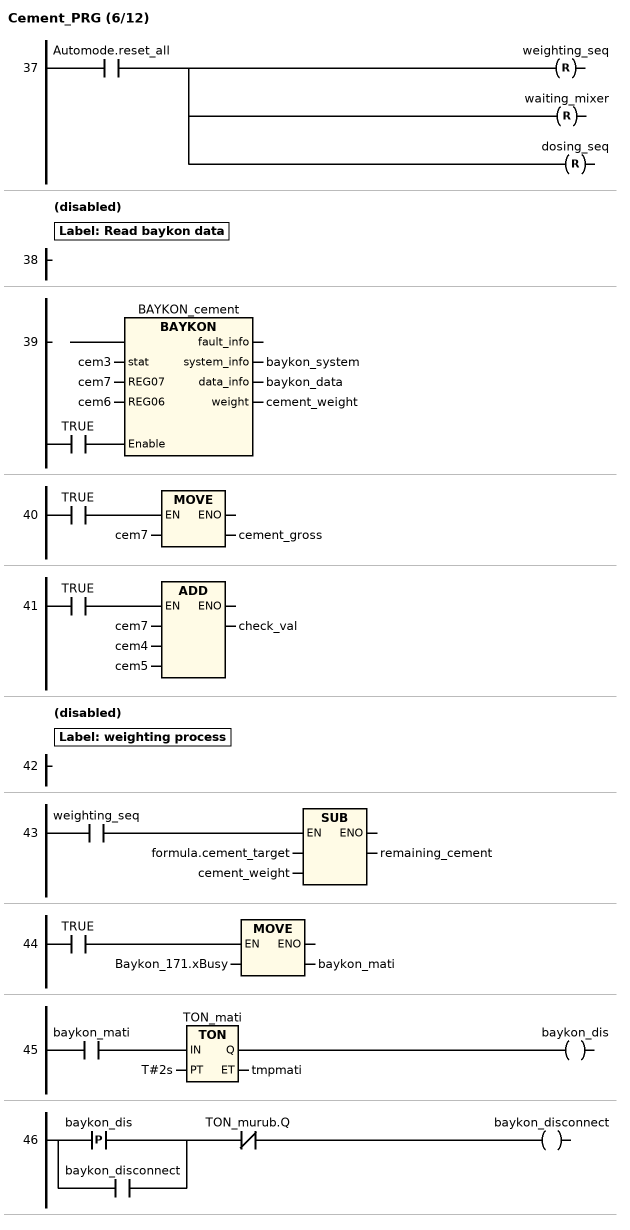
// NETWORK 37
weighting_seq R= Automode.reset_all;
waiting_mixer R= Automode.reset_all;
dosing_seq R= Automode.reset_all;

// NETWORK 38 (disabled)
// label: Label: Read baykon data

// NETWORK 39
BAYKON_cement(
    stat := cem3,
    REG07 := cem7,
    REG06 := cem6,
    Enable := TRUE,
    system_info => baykon_system,
    data_info => baykon_data,
    weight => cement_weight); // BAYKON

// NETWORK 40
cement_gross := cem7;

// NETWORK 41
check_val := cem7 + cem4 + cem5;

// NETWORK 42 (disabled)
// label: Label: weighting process

// NETWORK 43
IF weighting_seq THEN remaining_cement := formula.cement_target - cement_weight; END_IF

// NETWORK 44
baykon_mati := Baykon_171.xBusy;

// NETWORK 45
TON_mati(IN := baykon_mati, PT := T#2s, ET => tmpmati); // TON
baykon_dis := TON_mati.Q;

// NETWORK 46
_rt13(CLK := baykon_dis);
baykon_disconnect := (_rt13.Q OR baykon_disconnect) AND NOT TON_murub.Q;

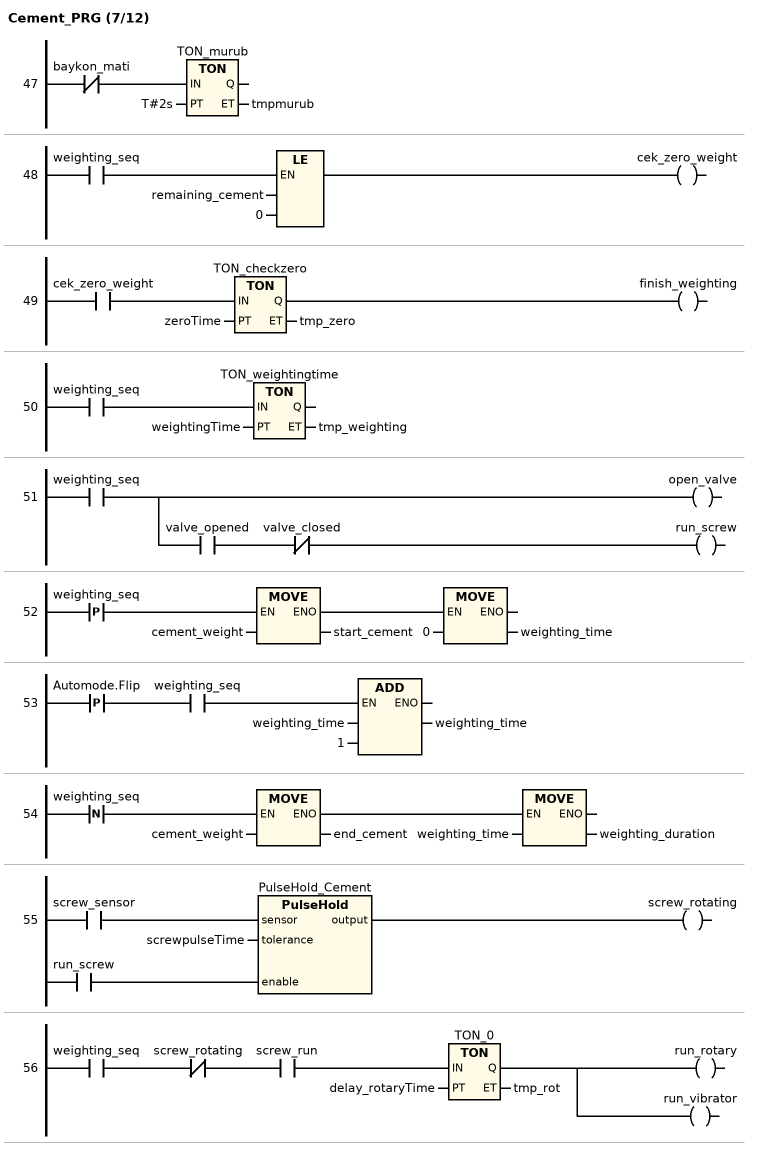
// NETWORK 47
TON_murub(IN := NOT baykon_mati, PT := T#2s, ET => tmpmurub); // TON

// NETWORK 48
cek_zero_weight := weighting_seq AND remaining_cement <= 0;

// NETWORK 49
TON_checkzero(IN := cek_zero_weight, PT := zeroTime, ET => tmp_zero); // TON
finish_weighting := TON_checkzero.Q;

// NETWORK 50
TON_weightingtime(IN := weighting_seq, PT := weightingTime, ET => tmp_weighting); // TON

// NETWORK 51
open_valve := weighting_seq;
run_screw := weighting_seq AND valve_opened AND NOT valve_closed;

// NETWORK 52
_rt14(CLK := weighting_seq);
_w4 := _rt14.Q;
IF _w4 THEN start_cement := cement_weight; END_IF
IF _w4 THEN weighting_time := 0; END_IF

// NETWORK 53
_rt15(CLK := Automode.Flip);
IF _rt15.Q AND weighting_seq THEN weighting_time := weighting_time + 1; END_IF

// NETWORK 54
_ft1(CLK := weighting_seq);
_w5 := _ft1.Q;
IF _w5 THEN end_cement := cement_weight; END_IF
IF _w5 THEN weighting_duration := weighting_time; END_IF

// NETWORK 55
PulseHold_Cement(sensor := screw_sensor, tolerance := screwpulseTime, enable := run_screw); // PulseHold
screw_rotating := PulseHold_Cement.output;

// NETWORK 56
TON_0(IN := weighting_seq AND NOT screw_rotating AND screw_run, PT := delay_rotaryTime, ET => tmp_rot); // TON
run_rotary := TON_0.Q;
run_vibrator := TON_0.Q;

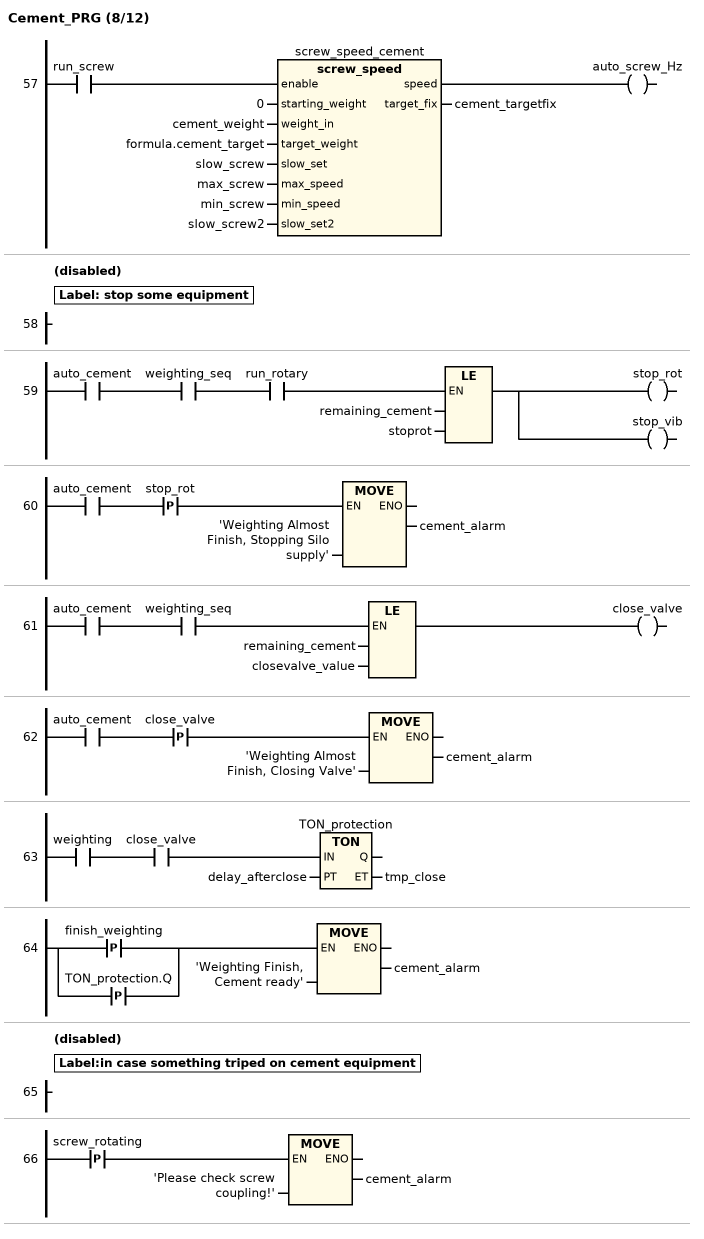
// NETWORK 57
screw_speed_cement(
    enable := run_screw,
    starting_weight := 0,
    weight_in := cement_weight,
    target_weight := formula.cement_target,
    slow_set := slow_screw,
    max_speed := max_screw,
    min_speed := min_screw,
    slow_set2 := slow_screw2,
    target_fix => cement_targetfix); // screw_speed
auto_screw_Hz := screw_speed_cement.speed;

// NETWORK 58 (disabled)
// label: Label: stop some equipment

// NETWORK 59
_w6 := auto_cement AND weighting_seq AND run_rotary AND remaining_cement <= stoprot;
stop_rot := _w6;
stop_vib := _w6;

// NETWORK 60
_rt16(CLK := stop_rot);
IF auto_cement AND _rt16.Q THEN cement_alarm := 'Weighting Almost Finish, Stopping Silo supply'; END_IF

// NETWORK 61
close_valve := auto_cement AND weighting_seq AND remaining_cement <= closevalve_value;

// NETWORK 62
_rt17(CLK := close_valve);
IF auto_cement AND _rt17.Q THEN cement_alarm := 'Weighting Almost Finish, Closing Valve'; END_IF

// NETWORK 63
TON_protection(IN := weighting AND close_valve, PT := delay_afterclose, ET => tmp_close); // TON

// NETWORK 64
_rt18(CLK := finish_weighting);
_rt19(CLK := TON_protection.Q);
IF _rt18.Q OR _rt19.Q THEN cement_alarm := 'Weighting Finish, Cement ready'; END_IF

// NETWORK 65 (disabled)
// label: Label:in case something triped on cement equipment

// NETWORK 66
_rt20(CLK := screw_rotating);
IF _rt20.Q THEN cement_alarm := 'Please check screw coupling!'; END_IF

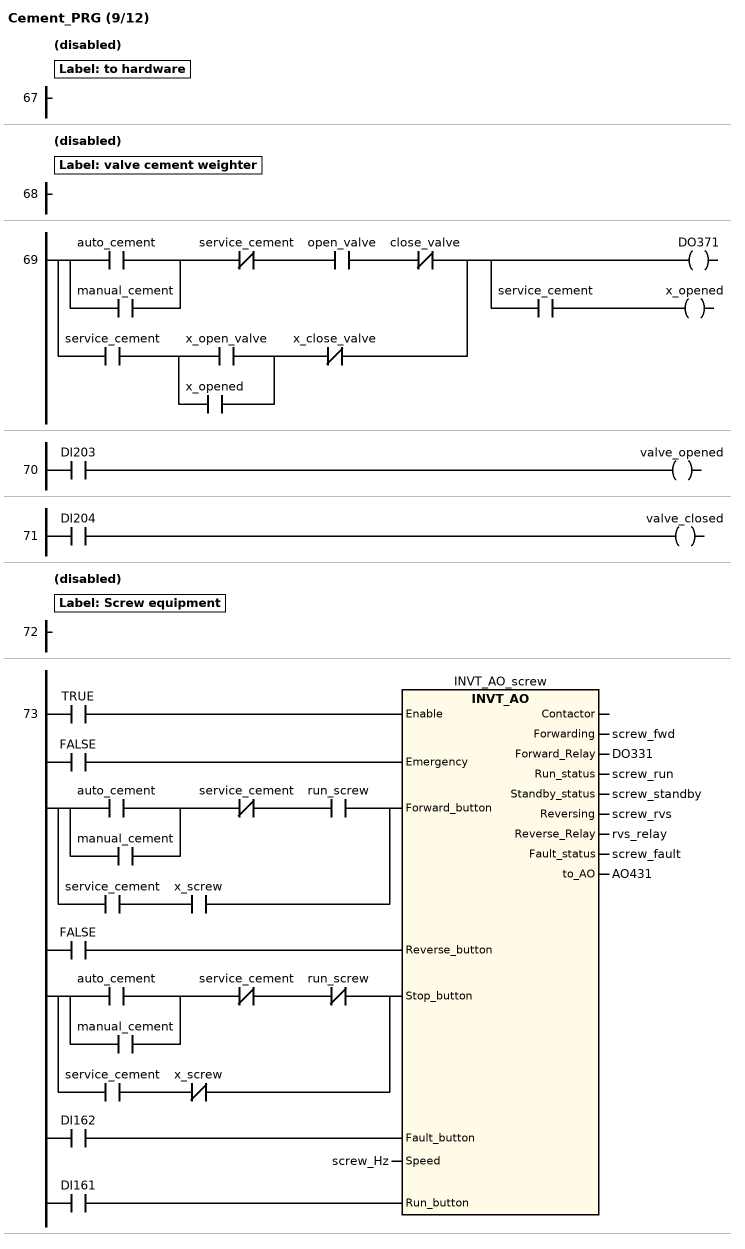
// NETWORK 67 (disabled)
// label: Label: to hardware

// NETWORK 68 (disabled)
// label: Label: valve cement weighter

// NETWORK 69
_w7 := (auto_cement OR manual_cement) AND NOT service_cement AND open_valve AND NOT close_valve OR service_cement AND (x_open_valve OR x_opened) AND NOT x_close_valve;
DO371 := _w7;
x_opened := _w7 AND service_cement;

// NETWORK 70
valve_opened := DI203;

// NETWORK 71
valve_closed := DI204;

// NETWORK 72 (disabled)
// label: Label: Screw equipment

// NETWORK 73
INVT_AO_screw(
    Enable := TRUE,
    Emergency := FALSE,
    Forward_button := (auto_cement OR manual_cement) AND NOT service_cement AND run_screw OR service_cement AND x_screw,
    Reverse_button := FALSE,
    Stop_button := (auto_cement OR manual_cement) AND NOT service_cement AND NOT run_screw OR service_cement AND NOT x_screw,
    Fault_button := DI162,
    Speed := screw_Hz,
    Run_button := DI161,
    Forwarding => screw_fwd,
    Forward_Relay => DO331,
    Run_status => screw_run,
    Standby_status => screw_standby,
    Reversing => screw_rvs,
    Reverse_Relay => rvs_relay,
    Fault_status => screw_fault,
    to_AO => AO431); // INVT_AO

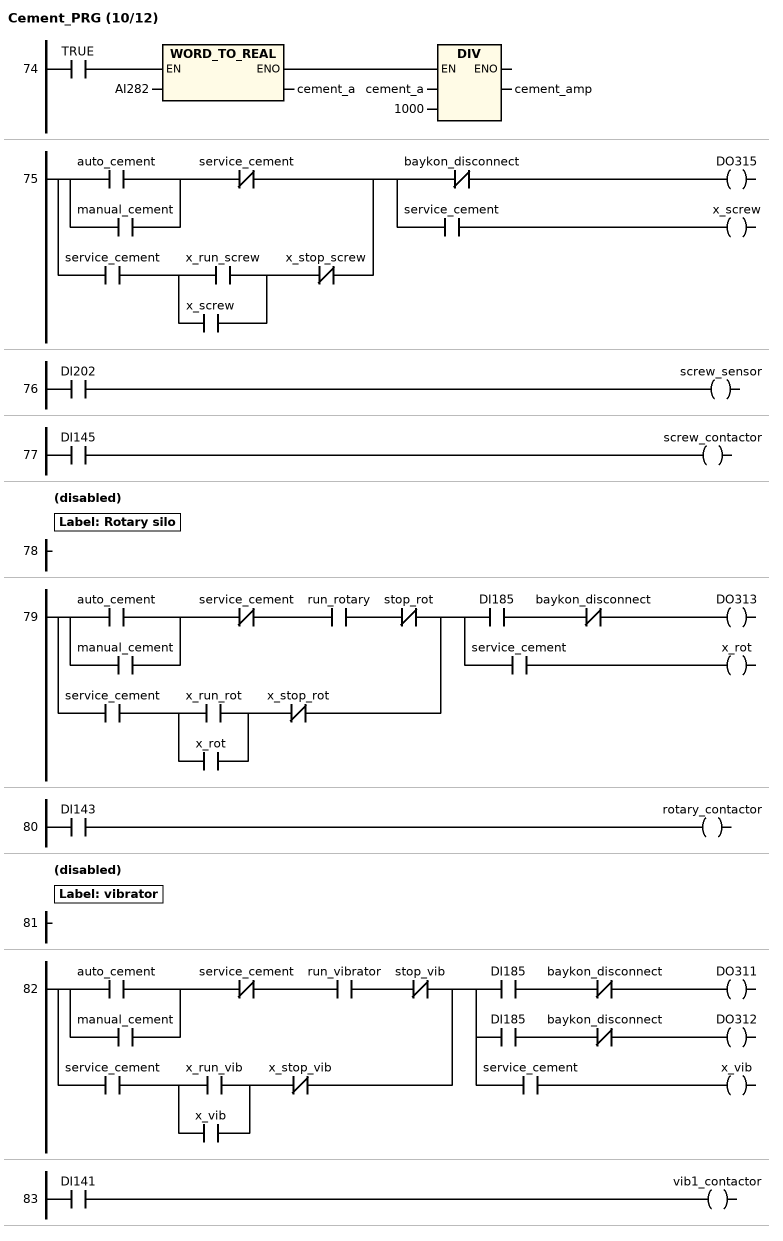
// NETWORK 74
cement_a := WORD_TO_REAL(AI282);
cement_amp := cement_a / 1000;

// NETWORK 75
_w8 := (auto_cement OR manual_cement) AND NOT service_cement OR service_cement AND (x_run_screw OR x_screw) AND NOT x_stop_screw;
DO315 := _w8 AND NOT baykon_disconnect;
x_screw := _w8 AND service_cement;

// NETWORK 76
screw_sensor := DI202;

// NETWORK 77
screw_contactor := DI145;

// NETWORK 78 (disabled)
// label: Label: Rotary silo

// NETWORK 79
_w9 := (auto_cement OR manual_cement) AND NOT service_cement AND run_rotary AND NOT stop_rot OR service_cement AND (x_run_rot OR x_rot) AND NOT x_stop_rot;
DO313 := _w9 AND DI185 AND NOT baykon_disconnect;
x_rot := _w9 AND service_cement;

// NETWORK 80
rotary_contactor := DI143;

// NETWORK 81 (disabled)
// label: Label: vibrator

// NETWORK 82
_w10 := (auto_cement OR manual_cement) AND NOT service_cement AND run_vibrator AND NOT stop_vib OR service_cement AND (x_run_vib OR x_vib) AND NOT x_stop_vib;
DO311 := _w10 AND DI185 AND NOT baykon_disconnect;
DO312 := _w10 AND DI185 AND NOT baykon_disconnect;
x_vib := _w10 AND service_cement;

// NETWORK 83
vib1_contactor := DI141;

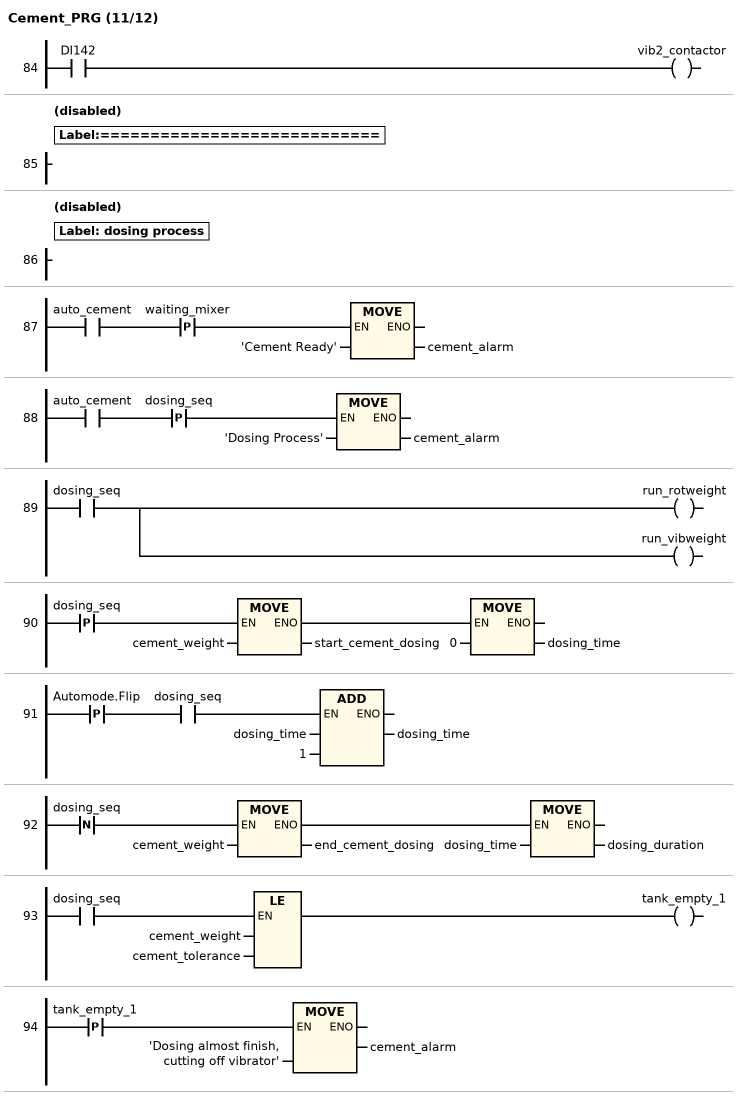
// NETWORK 84
vib2_contactor := DI142;

// NETWORK 85 (disabled)
// label: Label:============================

// NETWORK 86 (disabled)
// label: Label: dosing process

// NETWORK 87
_rt21(CLK := waiting_mixer);
IF auto_cement AND _rt21.Q THEN cement_alarm := 'Cement Ready'; END_IF

// NETWORK 88
_rt22(CLK := dosing_seq);
IF auto_cement AND _rt22.Q THEN cement_alarm := 'Dosing Process'; END_IF

// NETWORK 89
run_rotweight := dosing_seq;
run_vibweight := dosing_seq;

// NETWORK 90
_rt23(CLK := dosing_seq);
_w11 := _rt23.Q;
IF _w11 THEN start_cement_dosing := cement_weight; END_IF
IF _w11 THEN dosing_time := 0; END_IF

// NETWORK 91
_rt24(CLK := Automode.Flip);
IF _rt24.Q AND dosing_seq THEN dosing_time := dosing_time + 1; END_IF

// NETWORK 92
_ft2(CLK := dosing_seq);
_w12 := _ft2.Q;
IF _w12 THEN end_cement_dosing := cement_weight; END_IF
IF _w12 THEN dosing_duration := dosing_time; END_IF

// NETWORK 93
tank_empty_1 := dosing_seq AND cement_weight <= cement_tolerance;

// NETWORK 94
_rt25(CLK := tank_empty_1);
IF _rt25.Q THEN cement_alarm := 'Dosing almost finish, cutting off vibrator'; END_IF

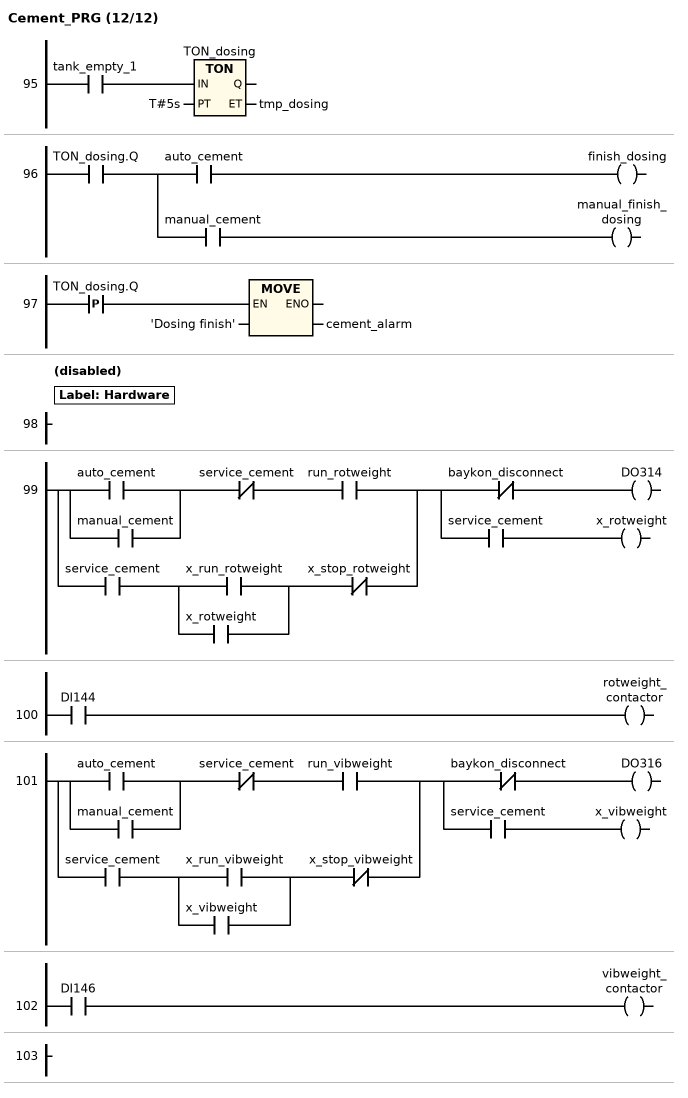
// NETWORK 95
TON_dosing(IN := tank_empty_1, PT := T#5s, ET => tmp_dosing); // TON

// NETWORK 96
finish_dosing := TON_dosing.Q AND auto_cement;
manual_finish_dosing := TON_dosing.Q AND manual_cement;

// NETWORK 97
_rt26(CLK := TON_dosing.Q);
IF _rt26.Q THEN cement_alarm := 'Dosing finish'; END_IF

// NETWORK 98 (disabled)
// label: Label: Hardware

// NETWORK 99
_w13 := (auto_cement OR manual_cement) AND NOT service_cement AND run_rotweight OR service_cement AND (x_run_rotweight OR x_rotweight) AND NOT x_stop_rotweight;
DO314 := _w13 AND NOT baykon_disconnect;
x_rotweight := _w13 AND service_cement;

// NETWORK 100
rotweight_contactor := DI144;

// NETWORK 101
_w14 := (auto_cement OR manual_cement) AND NOT service_cement AND run_vibweight OR service_cement AND (x_run_vibweight OR x_vibweight) AND NOT x_stop_vibweight;
DO316 := _w14 AND NOT baykon_disconnect;
x_vibweight := _w14 AND service_cement;

// NETWORK 102
vibweight_contactor := DI146;

// NETWORK 103

END_PROGRAM

// Device/Application/Automode
PROGRAM Automode
VAR
	run_batch: BOOL;
	enable: BOOL;
	finish_batch: BOOL;
	last_batch: BOOL;
	end_batch: BOOL;
	disable: BOOL;
	interupt_0: interupt;
	mortar_ready: BOOL;
	
	lime_setpoint: REAL;
	cement_setpoint: REAL;
	mixer_ready: BOOL;
	run_all: BOOL;
	cement_ready: BOOL;
	dose_cement_ready: BOOL;
	show_start: BOOL;
	is_mixer_empty: BOOL;
	mixer_empty: BOOL;
	mixer_full: BOOL;
	dosing_request: BOOL;
	dosing_finish: BOOL;
	mixing_process: BOOL;
	TON_flip: TON;
	TON_flop: TON;
	Flip: BOOL;
	tmp_flip: TIME;
	tmp_flop: TIME;
	TON_flick: TON;
	TON_flock: TON;
	tmp_flick: TIME;
	tmp_flock: TIME;
	Flick: BOOL;
	ParamAdjust_interval: ParamAdjust;
	// s
	interval: REAL := 180;
	add_interval: BOOL;
	sub_interval: BOOL;
	intervalms: REAL;
	intervalTime: TIME;
	ParamAdjust_distance: ParamAdjust;
	// s
	distance: REAL := 10;
	distancems: REAL;
	distanceTime: TIME;
	ParamAdjust_pulse: ParamAdjust;
	// ms
	pulse: REAL := 300;
	add_distance: BOOL;
	sub_distance: BOOL;
	add_pulse: BOOL;
	sub_pulse: BOOL;
	pulseTime: TIME;
	auto_dust: BOOL;
	manual_dust: BOOL;
	TON_start: TON;
	tmp_start: TIME;
	auto_packing: BOOL;
	auto_mode: BOOL;
	lime_ready: BOOL;
	DC_0: DC;
	dc_signal: WORD;
	Runbelt: BOOL;
	mixer_finish: BOOL;
	mixend: BOOL;
	disable_cement: BOOL;
	lime_dosing_finish: BOOL;
	cement_dosing_finish: BOOL;
	log_mortar: BOOL;
	start_cement: REAL;
	end_cement: REAL;
	weighting_duration: INT;
	dust_col_run: BOOL;
	reset_all: BOOL;
	last_load: BOOL;
	teslog: BOOL;
	jepit: BOOL;
	release: BOOL;
	tembak: BOOL;
	TON_0: TON;
	variable: TIME;
	tendang: BOOL;
	TON_1: TON;
	T3s: TIME;
	ter: TIME;
	TOF_1: TOF;
	relase: BOOL;
	t: BOOL;
	TON_2: TON;
	TOF_0: TOF;
	TON_3: TON;
	TON_4: TON;
	tmpx3: TIME;
	tmpx4: TIME;
END_VAR
VAR // added by the converter: edge detectors and wires of the graphical bodies
    _w1, _w2, _w3 : BOOL;
    _rt1, _rt2, _rt3, _rt4, _rt5 : R_TRIG;
    _ft1, _ft2, _ft3 : F_TRIG;
END_VAR

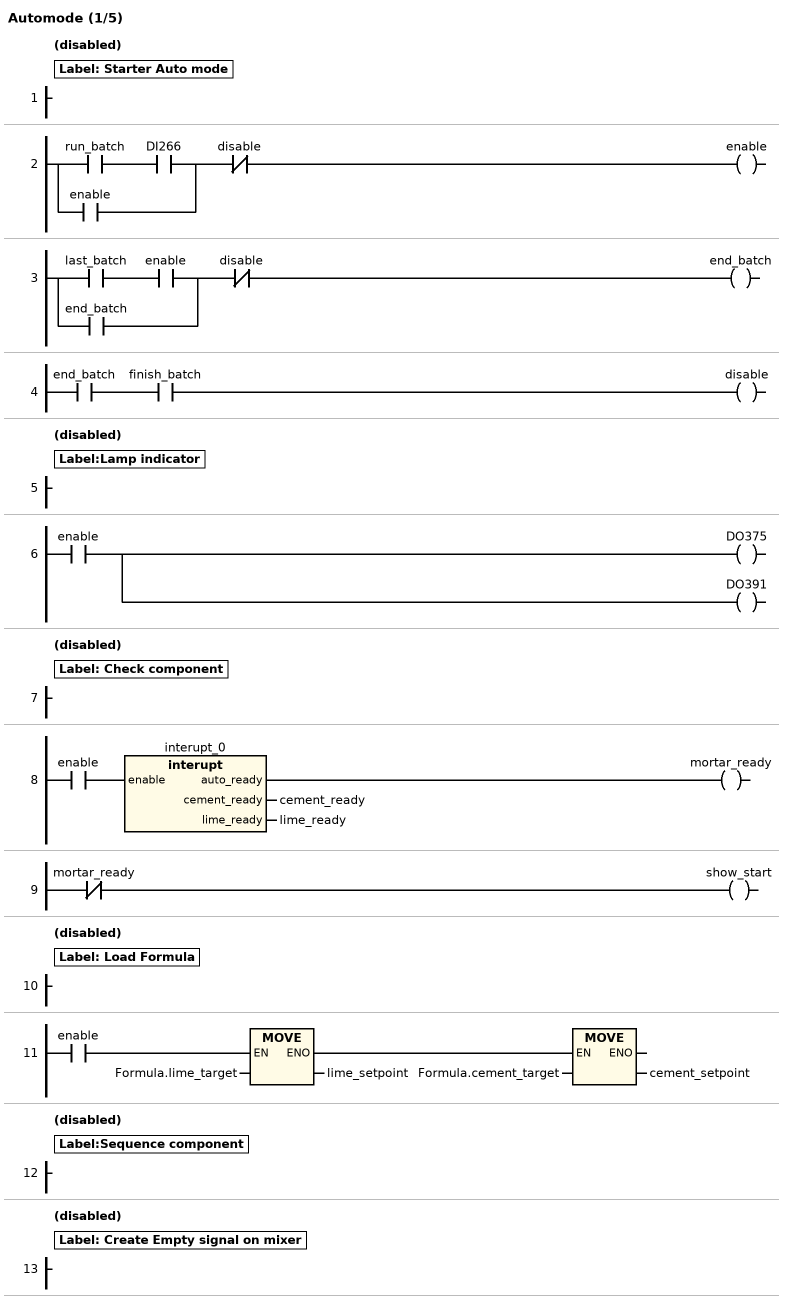
// NETWORK 1 (disabled)
// label: Label: Starter Auto mode

// NETWORK 2
enable := (run_batch AND DI266 OR enable) AND NOT disable;

// NETWORK 3
end_batch := (last_batch AND enable OR end_batch) AND NOT disable;

// NETWORK 4
disable := end_batch AND finish_batch;

// NETWORK 5 (disabled)
// label: Label:Lamp indicator

// NETWORK 6
DO375 := enable;
DO391 := enable;

// NETWORK 7 (disabled)
// label: Label: Check component

// NETWORK 8
interupt_0(enable := enable, cement_ready => cement_ready, lime_ready => lime_ready); // interupt
mortar_ready := interupt_0.auto_ready;

// NETWORK 9
show_start := NOT mortar_ready;

// NETWORK 10 (disabled)
// label: Label: Load Formula

// NETWORK 11
_w1 := enable;
IF _w1 THEN lime_setpoint := Formula.lime_target; END_IF
IF _w1 THEN cement_setpoint := Formula.cement_target; END_IF

// NETWORK 12 (disabled)
// label: Label:Sequence component

// NETWORK 13 (disabled)
// label: Label: Create Empty signal on mixer

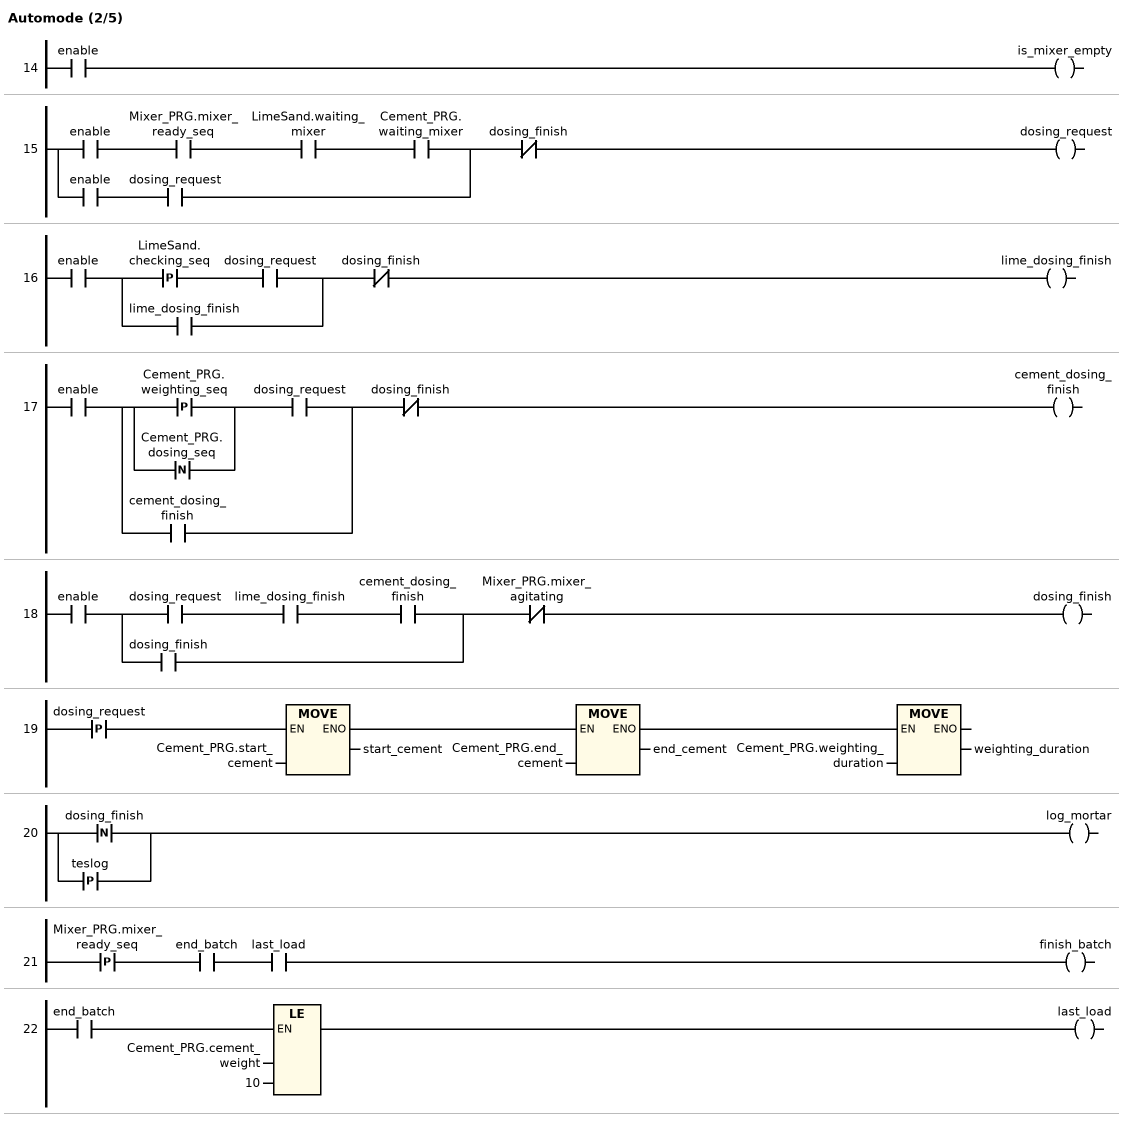
// NETWORK 14
is_mixer_empty := enable;

// NETWORK 15
dosing_request := (enable AND Mixer_PRG.mixer_ready_seq AND LimeSand.waiting_mixer AND Cement_PRG.waiting_mixer OR enable AND dosing_request) AND NOT dosing_finish;

// NETWORK 16
_rt1(CLK := LimeSand.checking_seq);
lime_dosing_finish := enable AND (_rt1.Q AND dosing_request OR lime_dosing_finish) AND NOT dosing_finish;

// NETWORK 17
_rt2(CLK := Cement_PRG.weighting_seq);
_ft1(CLK := Cement_PRG.dosing_seq);
cement_dosing_finish := enable AND ((_rt2.Q OR _ft1.Q) AND dosing_request OR cement_dosing_finish) AND NOT dosing_finish;

// NETWORK 18
dosing_finish := enable AND (dosing_request AND lime_dosing_finish AND cement_dosing_finish OR dosing_finish) AND NOT Mixer_PRG.mixer_agitating;

// NETWORK 19
_rt3(CLK := dosing_request);
_w2 := _rt3.Q;
IF _w2 THEN start_cement := Cement_PRG.start_cement; END_IF
IF _w2 THEN end_cement := Cement_PRG.end_cement; END_IF
IF _w2 THEN weighting_duration := Cement_PRG.weighting_duration; END_IF

// NETWORK 20
_ft2(CLK := dosing_finish);
_rt4(CLK := teslog);
log_mortar := _ft2.Q OR _rt4.Q;

// NETWORK 21
_rt5(CLK := Mixer_PRG.mixer_ready_seq);
finish_batch := _rt5.Q AND end_batch AND last_load;

// NETWORK 22
last_load := end_batch AND Cement_PRG.cement_weight <= 10;

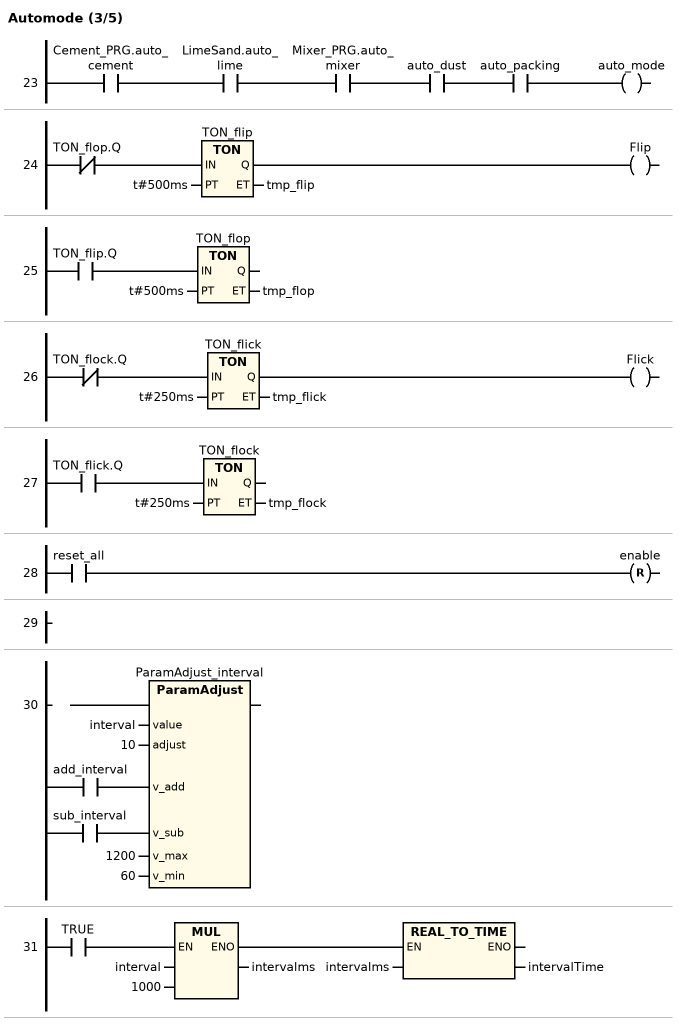
// NETWORK 23
auto_mode := Cement_PRG.auto_cement AND LimeSand.auto_lime AND Mixer_PRG.auto_mixer AND auto_dust AND auto_packing;

// NETWORK 24
TON_flip(IN := NOT TON_flop.Q, PT := t#500ms, ET => tmp_flip); // TON
Flip := TON_flip.Q;

// NETWORK 25
TON_flop(IN := TON_flip.Q, PT := t#500ms, ET => tmp_flop); // TON

// NETWORK 26
TON_flick(IN := NOT TON_flock.Q, PT := t#250ms, ET => tmp_flick); // TON
Flick := TON_flick.Q;

// NETWORK 27
TON_flock(IN := TON_flick.Q, PT := t#250ms, ET => tmp_flock); // TON

// NETWORK 28
enable R= reset_all;

// NETWORK 29

// NETWORK 30
ParamAdjust_interval(
    value := interval,
    adjust := 10,
    v_add := add_interval,
    v_sub := sub_interval,
    v_max := 1200,
    v_min := 60); // ParamAdjust

// NETWORK 31
intervalms := interval * 1000;
intervalTime := REAL_TO_TIME(intervalms);

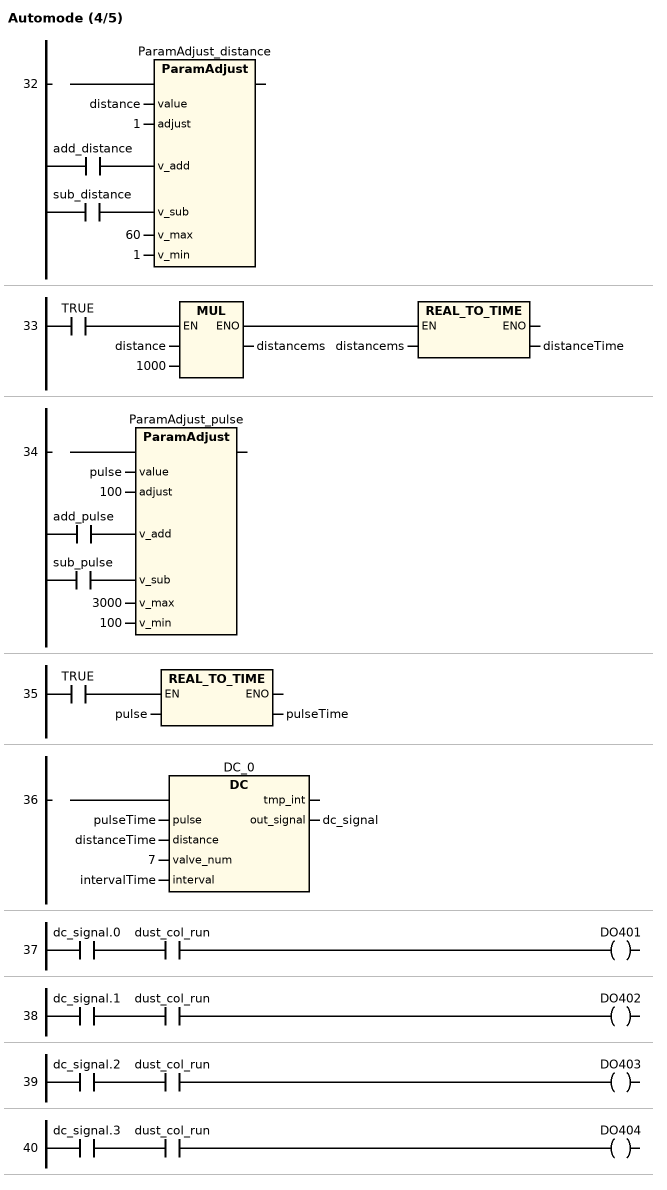
// NETWORK 32
ParamAdjust_distance(
    value := distance,
    adjust := 1,
    v_add := add_distance,
    v_sub := sub_distance,
    v_max := 60,
    v_min := 1); // ParamAdjust

// NETWORK 33
distancems := distance * 1000;
distanceTime := REAL_TO_TIME(distancems);

// NETWORK 34
ParamAdjust_pulse(
    value := pulse,
    adjust := 100,
    v_add := add_pulse,
    v_sub := sub_pulse,
    v_max := 3000,
    v_min := 100); // ParamAdjust

// NETWORK 35
pulseTime := REAL_TO_TIME(pulse);

// NETWORK 36
DC_0(
    pulse := pulseTime,
    distance := distanceTime,
    valve_num := 7,
    interval := intervalTime,
    out_signal => dc_signal); // DC

// NETWORK 37
DO401 := dc_signal.0 AND dust_col_run;

// NETWORK 38
DO402 := dc_signal.1 AND dust_col_run;

// NETWORK 39
DO403 := dc_signal.2 AND dust_col_run;

// NETWORK 40
DO404 := dc_signal.3 AND dust_col_run;

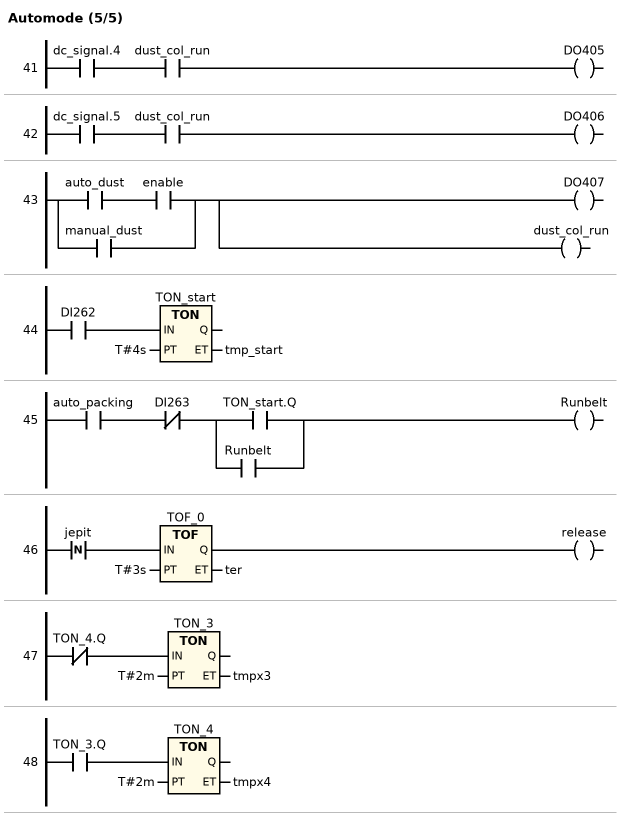
// NETWORK 41
DO405 := dc_signal.4 AND dust_col_run;

// NETWORK 42
DO406 := dc_signal.5 AND dust_col_run;

// NETWORK 43
_w3 := auto_dust AND enable OR manual_dust;
DO407 := _w3;
dust_col_run := _w3;

// NETWORK 44
TON_start(IN := DI262, PT := T#4s, ET => tmp_start); // TON

// NETWORK 45
Runbelt := auto_packing AND NOT DI263 AND (TON_start.Q OR Runbelt);

// NETWORK 46
_ft3(CLK := jepit);
TOF_0(IN := _ft3.Q, PT := T#3s, ET => ter); // TOF
release := TOF_0.Q;

// NETWORK 47
TON_3(IN := NOT TON_4.Q, PT := T#2m, ET => tmpx3); // TON

// NETWORK 48
TON_4(IN := TON_3.Q, PT := T#2m, ET => tmpx4); // TON

END_PROGRAM

// Device/Application/interupt
FUNCTION_BLOCK interupt
VAR_INPUT
	enable: BOOL;
END_VAR
VAR_OUTPUT
	auto_ready: BOOL;
	cement_ready: BOOL;
END_VAR
VAR
	mixer_ready: BOOL;
END_VAR
VAR_OUTPUT
	lime_ready: BOOL;
END_VAR
VAR
	power_ready: BOOL;
	LBcement_ready: BOOL;
	LBmixer_ready: BOOL;
	LBlime_ready: BOOL;
	mixer2_ready: BOOL;
	LBmixer2_ready: BOOL;
	Vib_cement: BOOL;
	Vib_mixer: BOOL;
	packing_ready: BOOL;
	Vib_lime: BOOL;
	Vib_sand: BOOL;
END_VAR

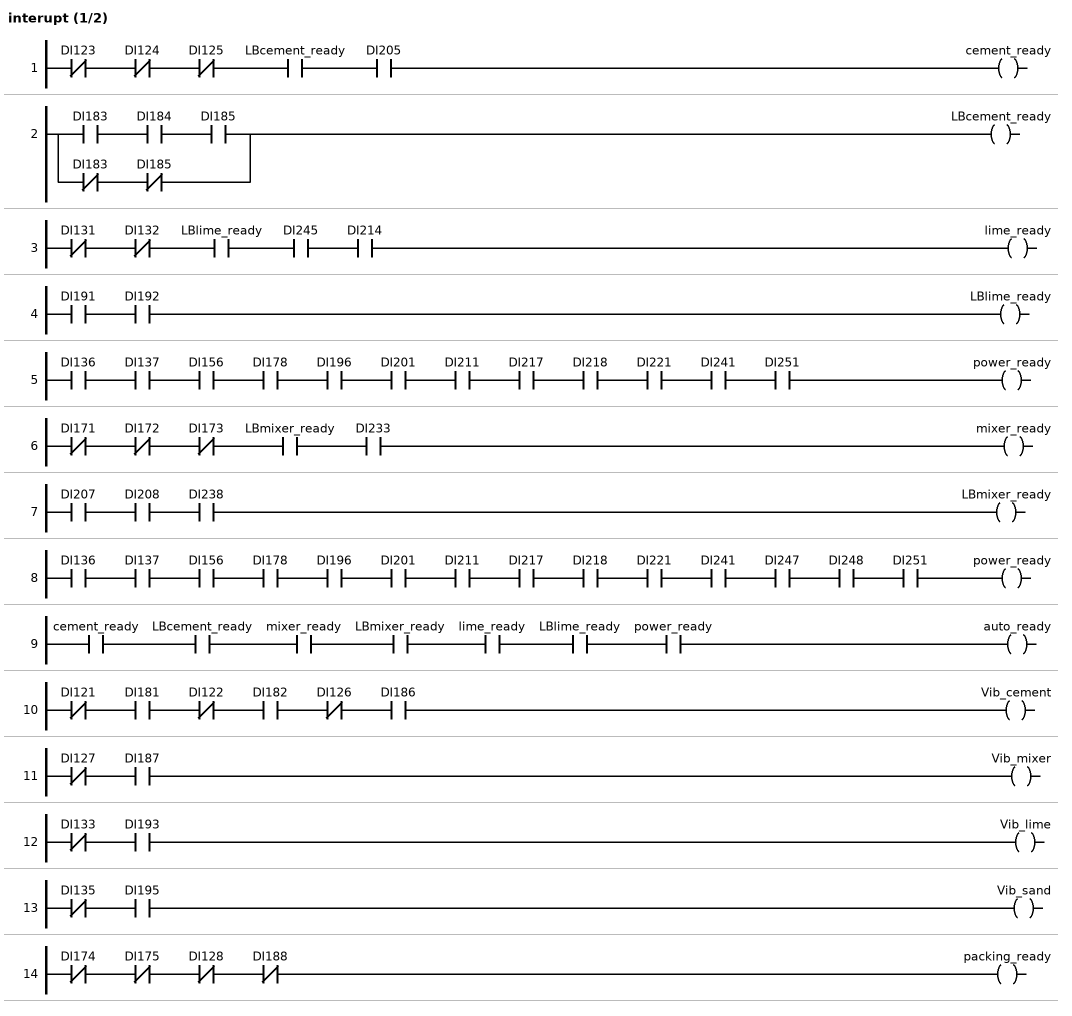
// NETWORK 1
cement_ready := NOT DI123 AND NOT DI124 AND NOT DI125 AND LBcement_ready AND DI205;

// NETWORK 2
LBcement_ready := DI183 AND DI184 AND DI185 OR NOT DI183 AND NOT DI185;

// NETWORK 3
lime_ready := NOT DI131 AND NOT DI132 AND LBlime_ready AND DI245 AND DI214;

// NETWORK 4
LBlime_ready := DI191 AND DI192;

// NETWORK 5
power_ready := DI136 AND DI137 AND DI156 AND DI178 AND DI196 AND DI201 AND DI211 AND DI217 AND DI218 AND DI221 AND DI241 AND DI251;

// NETWORK 6
mixer_ready := NOT DI171 AND NOT DI172 AND NOT DI173 AND LBmixer_ready AND DI233;

// NETWORK 7
LBmixer_ready := DI207 AND DI208 AND DI238;

// NETWORK 8
power_ready := DI136 AND DI137 AND DI156 AND DI178 AND DI196 AND DI201 AND DI211 AND DI217 AND DI218 AND DI221 AND DI241 AND DI247 AND DI248 AND DI251;

// NETWORK 9
auto_ready := cement_ready AND LBcement_ready AND mixer_ready AND LBmixer_ready AND lime_ready AND LBlime_ready AND power_ready;

// NETWORK 10
Vib_cement := NOT DI121 AND DI181 AND NOT DI122 AND DI182 AND NOT DI126 AND DI186;

// NETWORK 11
Vib_mixer := NOT DI127 AND DI187;

// NETWORK 12
Vib_lime := NOT DI133 AND DI193;

// NETWORK 13
Vib_sand := NOT DI135 AND DI195;

// NETWORK 14
packing_ready := NOT DI174 AND NOT DI175 AND NOT DI128 AND NOT DI188;

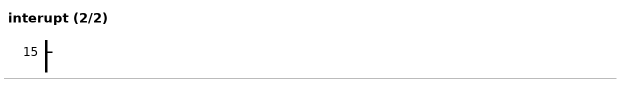
// NETWORK 15

END_FUNCTION_BLOCK

// Device/Application/Mixer_PRG
PROGRAM Mixer_PRG
VAR
	auto_mixer: BOOL;
	service_mixer: BOOL := true;
	manual_mixer: BOOL;
	x_run_mainagi: BOOL;
	interupted: BOOL;
	run_mainagi: BOOL;
	run_agi1: BOOL;
	run_agi2: BOOL;
	x_run_agi1: BOOL;
	x_run_agi2: BOOL;
	ParamAdjust_agitate: ParamAdjust;
	agitatedura: REAL := 200;
	add_agitatedura: BOOL;
	sub_agitatedura: BOOL;
	agitatedurams: REAL;
	agitateTime: TIME;
	manual_run_agitator: BOOL;
	run_agitator: BOOL;
	TON_agi: TON;
	tmp_agi: TIME;
	auto_mixerx: BOOL;
	manual_mixerx: BOOL;
	service_mixerx: BOOL;
	x_mainagi: BOOL;
	x_stop_mainagi: BOOL;
	x_stop_agi1: BOOL;
	x_agi1: BOOL;
	x_agi2: BOOL;
	x_stop_agi2: BOOL;
	manual_stop_agitator: BOOL;
	open_door: BOOL;
	x_open_door: BOOL;
	x_door_opened: BOOL;
	x_close_door: BOOL;
	start_blow: BOOL;
	x_start_blow: BOOL;
	x_blowing: BOOL;
	x_stop_blow: BOOL;
	contactor_mainagi: BOOL;
	contactor_mainagi_star: BOOL;
	contactor_mainagi_delta: BOOL;
	contactor_agi1: BOOL;
	contactor_agi2: BOOL;
	contactor_vibmixer: BOOL;
	run_vibrator: BOOL;
	x_run_vibmixer: BOOL;
	x_vibmixer: BOOL;
	x_stop_vibmixer: BOOL;
	run_beltpacking: BOOL;
	x_beltpacking: BOOL;
	x_run_beltpacking: BOOL;
	x_stop_beltpacking: BOOL;
	contactor_beltpacking: BOOL;
	empty_progress: BOOL;
	low_level: BOOL;
	med_level: BOOL;
	mixer_empty: BOOL;
	mixer_alarm: STRING;
	TON_empty: TON;
	ParamAdjust_Dosingtime: ParamAdjust;
	dosingtime: REAL := 15;
	add_dosingtime: BOOL;
	sub_dosingtime: BOOL;
	dosingtimems: REAL;
	dosingDelay: TIME;
	tmp_empty: TIME;
	mixer_full: BOOL;
	// PX sensor
	opened: BOOL;
	// RS sensor
	pneumatic_max: BOOL;
	mixer_ready: BOOL;
	// RS sensor
	pneumatic_min: BOOL;
	// PX sensor
	closed: BOOL;
	start_agitate: BOOL;
	dosing_to_hopper: BOOL;
	TON_agitating: TON;
	agi_ms: REAL;
	agiTime: TIME;
	tmp_agitate: TIME;
	mixer_waiting: BOOL;
	mixer_dosing: BOOL;
	dosing_finish: BOOL;
	check_ready: BOOL;
	mixer_ready_seq: BOOL;
	mixer_agitating: BOOL;
	agitating_finish: BOOL;
	mixer_seq: STRING;
END_VAR
VAR // added by the converter: edge detectors and wires of the graphical bodies
    _rt1, _rt2, _rt3, _rt4, _rt5, _rt6, _rt7, _rt8, _rt9, _rt10, _rt11, _rt12, _rt13, _rt14, _rt15, _rt16 : R_TRIG;
    _w1, _w2, _w3, _w4, _w5, _w6, _w7, _w8, _w9, _w10, _w11, _w12 : BOOL;
END_VAR

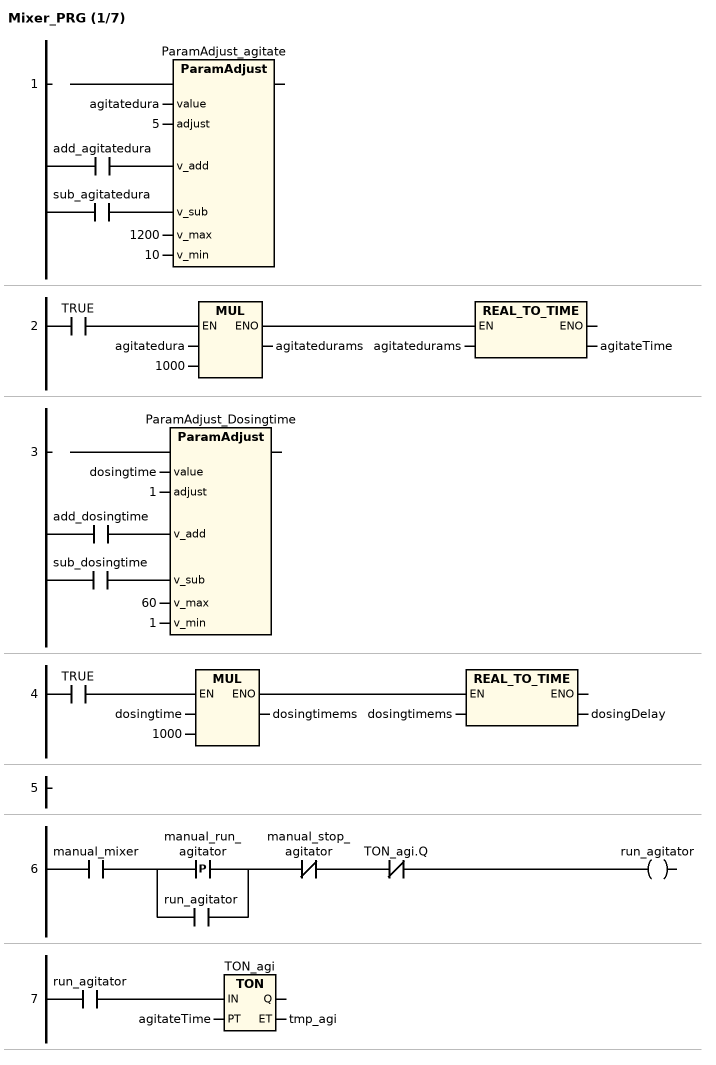
// NETWORK 1
ParamAdjust_agitate(
    value := agitatedura,
    adjust := 5,
    v_add := add_agitatedura,
    v_sub := sub_agitatedura,
    v_max := 1200,
    v_min := 10); // ParamAdjust

// NETWORK 2
agitatedurams := agitatedura * 1000;
agitateTime := REAL_TO_TIME(agitatedurams);

// NETWORK 3
ParamAdjust_Dosingtime(
    value := dosingtime,
    adjust := 1,
    v_add := add_dosingtime,
    v_sub := sub_dosingtime,
    v_max := 60,
    v_min := 1); // ParamAdjust

// NETWORK 4
dosingtimems := dosingtime * 1000;
dosingDelay := REAL_TO_TIME(dosingtimems);

// NETWORK 5

// NETWORK 6
_rt1(CLK := manual_run_agitator);
run_agitator := manual_mixer AND (_rt1.Q OR run_agitator) AND NOT manual_stop_agitator AND NOT TON_agi.Q;

// NETWORK 7
TON_agi(IN := run_agitator, PT := agitateTime, ET => tmp_agi); // TON

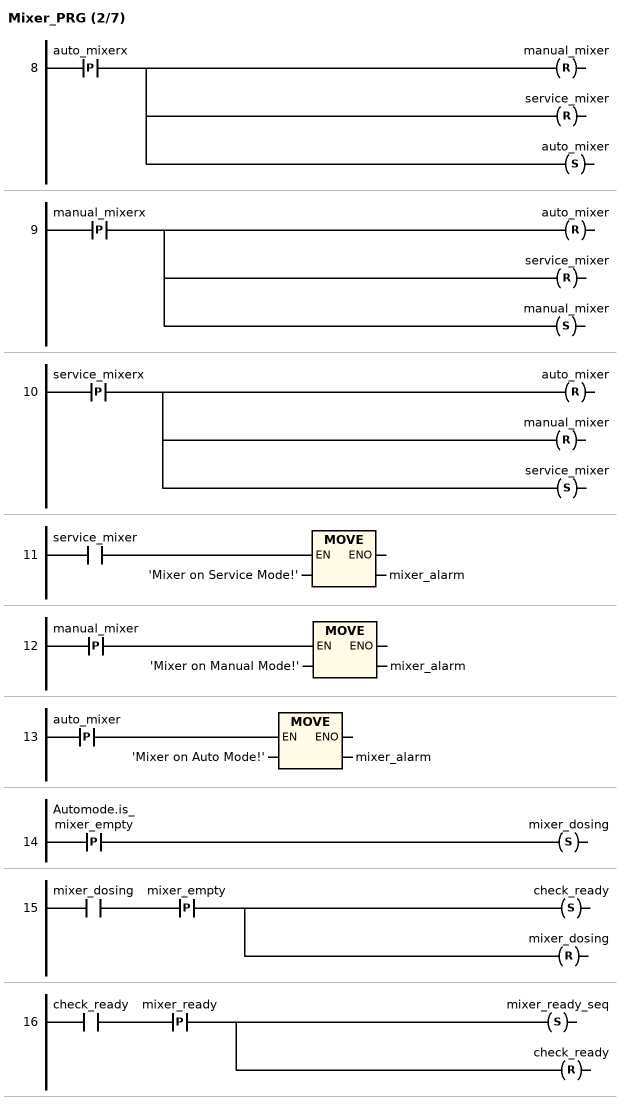
// NETWORK 8
_rt2(CLK := auto_mixerx);
manual_mixer R= _rt2.Q;
service_mixer R= _rt2.Q;
auto_mixer S= _rt2.Q;

// NETWORK 9
_rt3(CLK := manual_mixerx);
auto_mixer R= _rt3.Q;
service_mixer R= _rt3.Q;
manual_mixer S= _rt3.Q;

// NETWORK 10
_rt4(CLK := service_mixerx);
auto_mixer R= _rt4.Q;
manual_mixer R= _rt4.Q;
service_mixer S= _rt4.Q;

// NETWORK 11
IF service_mixer THEN mixer_alarm := 'Mixer on Service Mode!'; END_IF

// NETWORK 12
_rt5(CLK := manual_mixer);
IF _rt5.Q THEN mixer_alarm := 'Mixer on Manual Mode!'; END_IF

// NETWORK 13
_rt6(CLK := auto_mixer);
IF _rt6.Q THEN mixer_alarm := 'Mixer on Auto Mode!'; END_IF

// NETWORK 14
_rt7(CLK := Automode.is_mixer_empty);
mixer_dosing S= _rt7.Q;

// NETWORK 15
_rt8(CLK := mixer_empty);
_w1 := mixer_dosing AND _rt8.Q;
check_ready S= _w1;
mixer_dosing R= _w1;

// NETWORK 16
_rt9(CLK := mixer_ready);
_w2 := check_ready AND _rt9.Q;
mixer_ready_seq S= _w2;
check_ready R= _w2;

